REGION Network 82: [P4] Movimento BTRK da P3 Entry == a ==> P3 Exit == a ==> P3 to P4
   RUNG wire#powerrail
      Contact( #CIn.P3.Fermi.Rest )
      Contact( #Sts.P3.Fermi.Sens_Out )
      "BTrk_Presence"(Item := "BTrk".A0301."B"["BTRK_A0301_Pos3_Entry"])
      "BTrk_Absence"(Item := "BTrk".A0301."B"["BTRK_A0301_Pos3_Exit"])
      Move(in := "BTrk".A0301."B"["BTRK_A0301_Pos3_Entry"], out1 => "BTrk".A0301."B"["BTRK_A0301_Pos3_Exit"])
      "BTrk_Presence"(Item := "BTrk".A0301."B"["BTRK_A0301_Pos3_Exit"])
      Move(in := "BTrk".Empty, out1 => "BTrk".A0301."B"["BTRK_A0301_Pos3_Entry"])
   END_RUNG
   RUNG wire#powerrail
      Contact( "Sys".ByPass )
      Contact( #CIn.P3.Fermi.Rest )
      I_Contact( #Sts.P3.Fermi.Sens_Ing )
      I_Contact( #Sts.P3.Fermi.Sens_Out )
      "BTrk_Presence"(Item := "BTrk".A0301."B"["BTRK_A0301_Pos3_Entry"])
      "BTrk_Absence"(Item := "BTrk".A0301."B"["BTRK_A0301_Pos3_to_Pos4"])
      "BTrk_Absence"(Item := "BTrk".A0301."B"["BTRK_A0301_Pos4_Entry"])
      Move(in := "BTrk".A0301."B"["BTRK_A0301_Pos3_Entry"], out1 => "BTrk".A0301."B"["BTRK_A0301_Pos3_Exit"])
      "BTrk_Presence"(Item := "BTrk".A0301."B"["BTRK_A0301_Pos3_Exit"])
      Move(in := "BTrk".Empty, out1 => "BTrk".A0301."B"["BTRK_A0301_Pos3_Entry"])
   END_RUNG
   RUNG wire#powerrail
      Contact( #CIn.P3.Fermi.Rest )
      I_Contact( #Sts.P3.Fermi.Sens_Ing )
      I_Contact( #Sts.P3.Fermi.Sens_Out )
      "BTrk_Presence"(Item := "BTrk".A0301."B"["BTRK_A0301_Pos3_Exit"])
      Move(in := "BTrk".A0301."B"["BTRK_A0301_Pos3_Exit"], out1 => "BTrk".A0301."B"["BTRK_A0301_Pos3_to_Pos4"])
      "BTrk_Presence"(Item := "BTrk".A0301."B"["BTRK_A0301_Pos3_to_Pos4"])
      Move(in := "BTrk".Empty, out1 => "BTrk".A0301."B"["BTRK_A0301_Pos3_Exit"])
   END_RUNG
   // the same network as SCL:
   "BTrk_Presence"(EN := #CIn.P3.Fermi.Rest AND #Sts.P3.Fermi.Sens_Out,
                   Item := "BTrk".A0301."B"["BTRK_A0301_Pos3_Entry"],
                   ENO => #_w1);
   "BTrk_Absence"(EN := #_w1, Item := "BTrk".A0301."B"["BTRK_A0301_Pos3_Exit"], ENO => #_w2);
   IF #_w2 THEN
       "BTrk".A0301."B"["BTRK_A0301_Pos3_Exit"] := "BTrk".A0301."B"["BTRK_A0301_Pos3_Entry"];
   END_IF;
   "BTrk_Presence"(EN := #_w2, Item := "BTrk".A0301."B"["BTRK_A0301_Pos3_Exit"], ENO => #_w3);
   IF #_w3 THEN "BTrk".A0301."B"["BTRK_A0301_Pos3_Entry"] := "BTrk".Empty; END_IF;
   "BTrk_Presence"(EN := "Sys".ByPass AND #CIn.P3.Fermi.Rest AND NOT #Sts.P3.Fermi.Sens_Ing AND NOT #Sts.P3.Fermi.Sens_Out,
                   Item := "BTrk".A0301."B"["BTRK_A0301_Pos3_Entry"],
                   ENO => #_w4);
   "BTrk_Absence"(EN := #_w4, Item := "BTrk".A0301."B"["BTRK_A0301_Pos3_to_Pos4"], ENO => #_w5);
   "BTrk_Absence"(EN := #_w5, Item := "BTrk".A0301."B"["BTRK_A0301_Pos4_Entry"], ENO => #_w6);
   IF #_w6 THEN
       "BTrk".A0301."B"["BTRK_A0301_Pos3_Exit"] := "BTrk".A0301."B"["BTRK_A0301_Pos3_Entry"];
   END_IF;
   "BTrk_Presence"(EN := #_w6, Item := "BTrk".A0301."B"["BTRK_A0301_Pos3_Exit"], ENO => #_w7);
   IF #_w7 THEN "BTrk".A0301."B"["BTRK_A0301_Pos3_Entry"] := "BTrk".Empty; END_IF;
   "BTrk_Presence"(EN := #CIn.P3.Fermi.Rest AND NOT #Sts.P3.Fermi.Sens_Ing AND NOT #Sts.P3.Fermi.Sens_Out,
                   Item := "BTrk".A0301."B"["BTRK_A0301_Pos3_Exit"],
                   ENO => #_w8);
   IF #_w8 THEN
       "BTrk".A0301."B"["BTRK_A0301_Pos3_to_Pos4"] := "BTrk".A0301."B"["BTRK_A0301_Pos3_Exit"];
   END_IF;
   "BTrk_Presence"(EN := #_w8, Item := "BTrk".A0301."B"["BTRK_A0301_Pos3_to_Pos4"], ENO => #_w9);
   IF #_w9 THEN "BTrk".A0301."B"["BTRK_A0301_Pos3_Exit"] := "BTrk".Empty; END_IF;
END_REGION

REGION Network 83: [P4] Movimento BTRK da P3 a P4 == a ==> P4 Entry
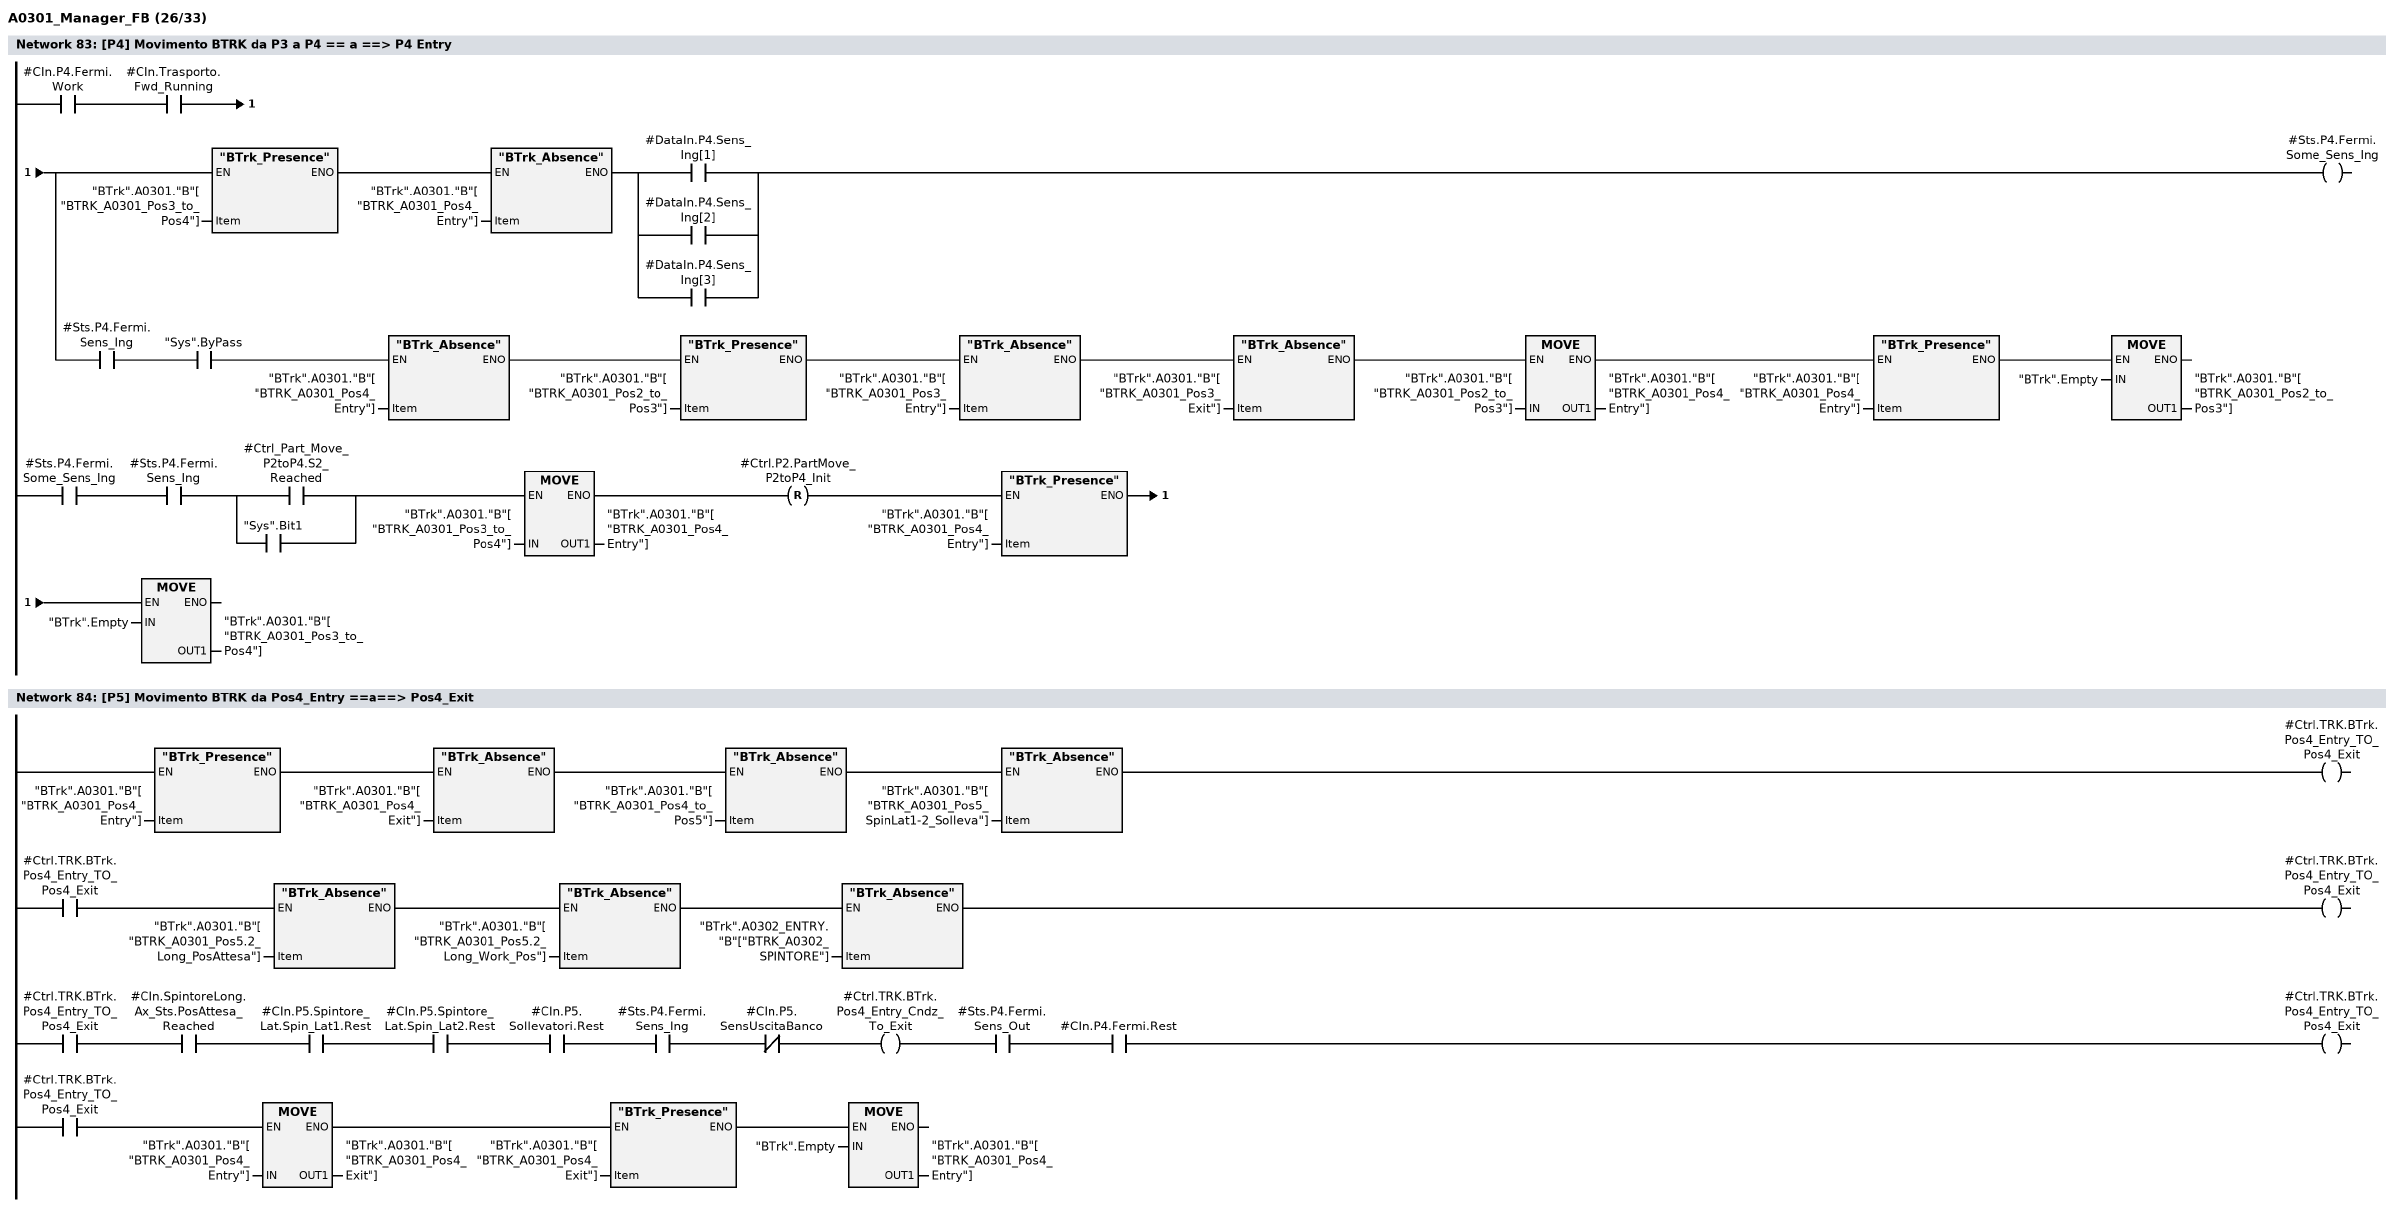
   RUNG wire#powerrail
      Contact( #CIn.P4.Fermi.Work )
      Contact( #CIn.Trasporto.Fwd_Running )
      wire#w1
      "BTrk_Presence"(Item := "BTrk".A0301."B"["BTRK_A0301_Pos3_to_Pos4"])
      "BTrk_Absence"(Item := "BTrk".A0301."B"["BTRK_A0301_Pos4_Entry"])
      wire#w2
      Contact( #DataIn.P4.Sens_Ing[1] )
      wire#w3
      Coil( #Sts.P4.Fermi.Some_Sens_Ing )
   END_RUNG
   RUNG wire#w2
      Contact( #DataIn.P4.Sens_Ing[2] )
   END_RUNG wire#w3
   RUNG wire#w2
      Contact( #DataIn.P4.Sens_Ing[3] )
   END_RUNG wire#w3
   RUNG wire#w1
      Contact( #Sts.P4.Fermi.Sens_Ing )
      Contact( "Sys".ByPass )
      "BTrk_Absence"(Item := "BTrk".A0301."B"["BTRK_A0301_Pos4_Entry"])
      "BTrk_Presence"(Item := "BTrk".A0301."B"["BTRK_A0301_Pos2_to_Pos3"])
      "BTrk_Absence"(Item := "BTrk".A0301."B"["BTRK_A0301_Pos3_Entry"])
      "BTrk_Absence"(Item := "BTrk".A0301."B"["BTRK_A0301_Pos3_Exit"])
      Move(in := "BTrk".A0301."B"["BTRK_A0301_Pos2_to_Pos3"], out1 => "BTrk".A0301."B"["BTRK_A0301_Pos4_Entry"])
      "BTrk_Presence"(Item := "BTrk".A0301."B"["BTRK_A0301_Pos4_Entry"])
      Move(in := "BTrk".Empty, out1 => "BTrk".A0301."B"["BTRK_A0301_Pos2_to_Pos3"])
   END_RUNG
   RUNG wire#powerrail
      Contact( #Sts.P4.Fermi.Some_Sens_Ing )
      Contact( #Sts.P4.Fermi.Sens_Ing )
      wire#w4
      Contact( #Ctrl_Part_Move_P2toP4.S2_Reached )
      wire#w5
      Move(in := "BTrk".A0301."B"["BTRK_A0301_Pos3_to_Pos4"], out1 => "BTrk".A0301."B"["BTRK_A0301_Pos4_Entry"])
      R_Coil( #Ctrl.P2.PartMove_P2toP4_Init )
      "BTrk_Presence"(Item := "BTrk".A0301."B"["BTRK_A0301_Pos4_Entry"])
      Move(in := "BTrk".Empty, out1 => "BTrk".A0301."B"["BTRK_A0301_Pos3_to_Pos4"])
   END_RUNG
   RUNG wire#w4
      Contact( "Sys".Bit1 )
   END_RUNG wire#w5
   // the same network as SCL:
   #_w1 := #CIn.P4.Fermi.Work AND #CIn.Trasporto.Fwd_Running;
   "BTrk_Presence"(EN := #_w1, Item := "BTrk".A0301."B"["BTRK_A0301_Pos3_to_Pos4"], ENO => #_w2);
   "BTrk_Absence"(EN := #_w2, Item := "BTrk".A0301."B"["BTRK_A0301_Pos4_Entry"], ENO => #_w3);
   #Sts.P4.Fermi.Some_Sens_Ing := #_w3 AND (#DataIn.P4.Sens_Ing[1] OR #DataIn.P4.Sens_Ing[2] OR #DataIn.P4.Sens_Ing[3]);
   "BTrk_Absence"(EN := #_w1 AND #Sts.P4.Fermi.Sens_Ing AND "Sys".ByPass,
                  Item := "BTrk".A0301."B"["BTRK_A0301_Pos4_Entry"],
                  ENO => #_w4);
   "BTrk_Presence"(EN := #_w4, Item := "BTrk".A0301."B"["BTRK_A0301_Pos2_to_Pos3"], ENO => #_w5);
   "BTrk_Absence"(EN := #_w5, Item := "BTrk".A0301."B"["BTRK_A0301_Pos3_Entry"], ENO => #_w6);
   "BTrk_Absence"(EN := #_w6, Item := "BTrk".A0301."B"["BTRK_A0301_Pos3_Exit"], ENO => #_w7);
   IF #_w7 THEN
       "BTrk".A0301."B"["BTRK_A0301_Pos4_Entry"] := "BTrk".A0301."B"["BTRK_A0301_Pos2_to_Pos3"];
   END_IF;
   "BTrk_Presence"(EN := #_w7, Item := "BTrk".A0301."B"["BTRK_A0301_Pos4_Entry"], ENO => #_w8);
   IF #_w8 THEN "BTrk".A0301."B"["BTRK_A0301_Pos2_to_Pos3"] := "BTrk".Empty; END_IF;
   IF #Sts.P4.Fermi.Some_Sens_Ing AND #Sts.P4.Fermi.Sens_Ing AND (#Ctrl_Part_Move_P2toP4.S2_Reached OR "Sys".Bit1) THEN
       "BTrk".A0301."B"["BTRK_A0301_Pos4_Entry"] := "BTrk".A0301."B"["BTRK_A0301_Pos3_to_Pos4"];
       #Ctrl.P2.PartMove_P2toP4_Init := FALSE;
   END_IF;
   "BTrk_Presence"(EN := #Sts.P4.Fermi.Some_Sens_Ing AND #Sts.P4.Fermi.Sens_Ing AND (#Ctrl_Part_Move_P2toP4.S2_Reached OR "Sys".Bit1),
                   Item := "BTrk".A0301."B"["BTRK_A0301_Pos4_Entry"],
                   ENO => #_w9);
   IF #_w9 THEN "BTrk".A0301."B"["BTRK_A0301_Pos3_to_Pos4"] := "BTrk".Empty; END_IF;
END_REGION

REGION Network 84: [P5] Movimento BTRK da Pos4_Entry ==a==> Pos4_Exit
   RUNG wire#powerrail
      "BTrk_Presence"(Item := "BTrk".A0301."B"["BTRK_A0301_Pos4_Entry"])
      "BTrk_Absence"(Item := "BTrk".A0301."B"["BTRK_A0301_Pos4_Exit"])
      "BTrk_Absence"(Item := "BTrk".A0301."B"["BTRK_A0301_Pos4_to_Pos5"])
      "BTrk_Absence"(Item := "BTrk".A0301."B"["BTRK_A0301_Pos5_SpinLat1-2_Solleva"])
      Coil( #Ctrl.TRK.BTrk.Pos4_Entry_TO_Pos4_Exit )
   END_RUNG
   RUNG wire#powerrail
      Contact( #Ctrl.TRK.BTrk.Pos4_Entry_TO_Pos4_Exit )
      "BTrk_Absence"(Item := "BTrk".A0301."B"["BTRK_A0301_Pos5.2_Long_PosAttesa"])
      "BTrk_Absence"(Item := "BTrk".A0301."B"["BTRK_A0301_Pos5.2_Long_Work_Pos"])
      "BTrk_Absence"(Item := "BTrk".A0302_ENTRY."B"["BTRK_A0302_SPINTORE"])
      Coil( #Ctrl.TRK.BTrk.Pos4_Entry_TO_Pos4_Exit )
   END_RUNG
   RUNG wire#powerrail
      Contact( #Ctrl.TRK.BTrk.Pos4_Entry_TO_Pos4_Exit )
      Contact( #CIn.SpintoreLong.Ax_Sts.PosAttesa_Reached )
      Contact( #CIn.P5.Spintore_Lat.Spin_Lat1.Rest )
      Contact( #CIn.P5.Spintore_Lat.Spin_Lat2.Rest )
      Contact( #CIn.P5.Sollevatori.Rest )
      Contact( #Sts.P4.Fermi.Sens_Ing )
      I_Contact( #CIn.P5.SensUscitaBanco )
      Coil( #Ctrl.TRK.BTrk.Pos4_Entry_Cndz_To_Exit )
      Contact( #Sts.P4.Fermi.Sens_Out )
      Contact( #CIn.P4.Fermi.Rest )
      Coil( #Ctrl.TRK.BTrk.Pos4_Entry_TO_Pos4_Exit )
   END_RUNG
   RUNG wire#powerrail
      Contact( #Ctrl.TRK.BTrk.Pos4_Entry_TO_Pos4_Exit )
      Move(in := "BTrk".A0301."B"["BTRK_A0301_Pos4_Entry"], out1 => "BTrk".A0301."B"["BTRK_A0301_Pos4_Exit"])
      "BTrk_Presence"(Item := "BTrk".A0301."B"["BTRK_A0301_Pos4_Exit"])
      Move(in := "BTrk".Empty, out1 => "BTrk".A0301."B"["BTRK_A0301_Pos4_Entry"])
   END_RUNG
   // the same network as SCL:
   "BTrk_Presence"(Item := "BTrk".A0301."B"["BTRK_A0301_Pos4_Entry"], ENO => #_w1);
   "BTrk_Absence"(EN := #_w1, Item := "BTrk".A0301."B"["BTRK_A0301_Pos4_Exit"], ENO => #_w2);
   "BTrk_Absence"(EN := #_w2, Item := "BTrk".A0301."B"["BTRK_A0301_Pos4_to_Pos5"], ENO => #_w3);
   "BTrk_Absence"(EN := #_w3, Item := "BTrk".A0301."B"["BTRK_A0301_Pos5_SpinLat1-2_Solleva"], ENO => #_w4);
   #Ctrl.TRK.BTrk.Pos4_Entry_TO_Pos4_Exit := #_w4;
   "BTrk_Absence"(EN := #Ctrl.TRK.BTrk.Pos4_Entry_TO_Pos4_Exit,
                  Item := "BTrk".A0301."B"["BTRK_A0301_Pos5.2_Long_PosAttesa"],
                  ENO => #_w5);
   "BTrk_Absence"(EN := #_w5, Item := "BTrk".A0301."B"["BTRK_A0301_Pos5.2_Long_Work_Pos"], ENO => #_w6);
   "BTrk_Absence"(EN := #_w6, Item := "BTrk".A0302_ENTRY."B"["BTRK_A0302_SPINTORE"], ENO => #_w7);
   #Ctrl.TRK.BTrk.Pos4_Entry_TO_Pos4_Exit := #_w7;
   #Ctrl.TRK.BTrk.Pos4_Entry_Cndz_To_Exit := #Ctrl.TRK.BTrk.Pos4_Entry_TO_Pos4_Exit AND #CIn.SpintoreLong.Ax_Sts.PosAttesa_Reached AND #CIn.P5.Spintore_Lat.Spin_Lat1.Rest AND #CIn.P5.Spintore_Lat.Spin_Lat2.Rest AND #CIn.P5.Sollevatori.Rest AND #Sts.P4.Fermi.Sens_Ing AND NOT #CIn.P5.SensUscitaBanco;
   #Ctrl.TRK.BTrk.Pos4_Entry_TO_Pos4_Exit := #Ctrl.TRK.BTrk.Pos4_Entry_Cndz_To_Exit AND #Sts.P4.Fermi.Sens_Out AND #CIn.P4.Fermi.Rest;
   IF #Ctrl.TRK.BTrk.Pos4_Entry_TO_Pos4_Exit THEN
       "BTrk".A0301."B"["BTRK_A0301_Pos4_Exit"] := "BTrk".A0301."B"["BTRK_A0301_Pos4_Entry"];
   END_IF;
   "BTrk_Presence"(EN := #Ctrl.TRK.BTrk.Pos4_Entry_TO_Pos4_Exit,
                   Item := "BTrk".A0301."B"["BTRK_A0301_Pos4_Exit"],
                   ENO => #_w8);
   IF #_w8 THEN "BTrk".A0301."B"["BTRK_A0301_Pos4_Entry"] := "BTrk".Empty; END_IF;
END_REGION

REGION Network 85: [P5] Movimento BTRK da Pos.4 Exit ==a==> Pos4_to_Pos5
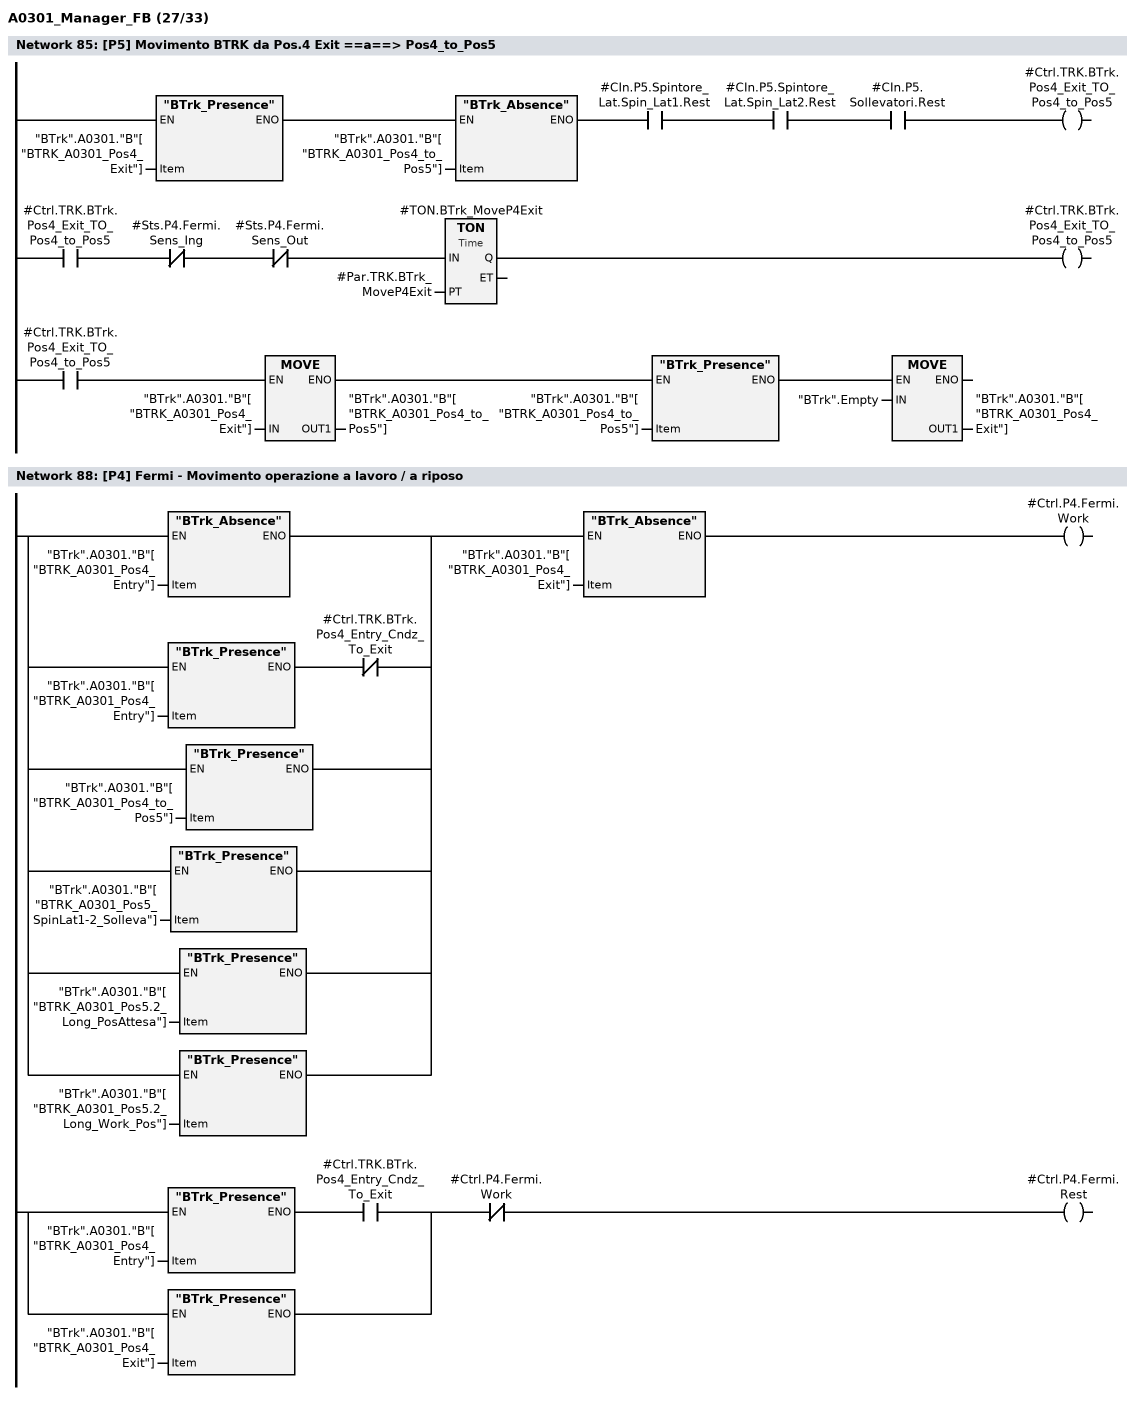
   RUNG wire#powerrail
      "BTrk_Presence"(Item := "BTrk".A0301."B"["BTRK_A0301_Pos4_Exit"])
      "BTrk_Absence"(Item := "BTrk".A0301."B"["BTRK_A0301_Pos4_to_Pos5"])
      Contact( #CIn.P5.Spintore_Lat.Spin_Lat1.Rest )
      Contact( #CIn.P5.Spintore_Lat.Spin_Lat2.Rest )
      Contact( #CIn.P5.Sollevatori.Rest )
      Coil( #Ctrl.TRK.BTrk.Pos4_Exit_TO_Pos4_to_Pos5 )
   END_RUNG
   RUNG wire#powerrail
      Contact( #Ctrl.TRK.BTrk.Pos4_Exit_TO_Pos4_to_Pos5 )
      I_Contact( #Sts.P4.Fermi.Sens_Ing )
      I_Contact( #Sts.P4.Fermi.Sens_Out )
      { S7_Templates := "time_type := Time" } #TON.BTrk_MoveP4Exit.TON(pt := #Par.TRK.BTrk_MoveP4Exit, et =>)
      Coil( #Ctrl.TRK.BTrk.Pos4_Exit_TO_Pos4_to_Pos5 )
   END_RUNG
   RUNG wire#powerrail
      Contact( #Ctrl.TRK.BTrk.Pos4_Exit_TO_Pos4_to_Pos5 )
      Move(in := "BTrk".A0301."B"["BTRK_A0301_Pos4_Exit"], out1 => "BTrk".A0301."B"["BTRK_A0301_Pos4_to_Pos5"])
      "BTrk_Presence"(Item := "BTrk".A0301."B"["BTRK_A0301_Pos4_to_Pos5"])
      Move(in := "BTrk".Empty, out1 => "BTrk".A0301."B"["BTRK_A0301_Pos4_Exit"])
   END_RUNG
   // the same network as SCL:
   "BTrk_Presence"(Item := "BTrk".A0301."B"["BTRK_A0301_Pos4_Exit"], ENO => #_w1);
   "BTrk_Absence"(EN := #_w1, Item := "BTrk".A0301."B"["BTRK_A0301_Pos4_to_Pos5"], ENO => #_w2);
   #Ctrl.TRK.BTrk.Pos4_Exit_TO_Pos4_to_Pos5 := #_w2 AND #CIn.P5.Spintore_Lat.Spin_Lat1.Rest AND #CIn.P5.Spintore_Lat.Spin_Lat2.Rest AND #CIn.P5.Sollevatori.Rest;
   #TON.BTrk_MoveP4Exit.TON(IN := #Ctrl.TRK.BTrk.Pos4_Exit_TO_Pos4_to_Pos5 AND NOT #Sts.P4.Fermi.Sens_Ing AND NOT #Sts.P4.Fermi.Sens_Out,
                           PT := #Par.TRK.BTrk_MoveP4Exit);
   #Ctrl.TRK.BTrk.Pos4_Exit_TO_Pos4_to_Pos5 := #TON.BTrk_MoveP4Exit.Q;
   IF #Ctrl.TRK.BTrk.Pos4_Exit_TO_Pos4_to_Pos5 THEN
       "BTrk".A0301."B"["BTRK_A0301_Pos4_to_Pos5"] := "BTrk".A0301."B"["BTRK_A0301_Pos4_Exit"];
   END_IF;
   "BTrk_Presence"(EN := #Ctrl.TRK.BTrk.Pos4_Exit_TO_Pos4_to_Pos5,
                   Item := "BTrk".A0301."B"["BTRK_A0301_Pos4_to_Pos5"],
                   ENO => #_w3);
   IF #_w3 THEN "BTrk".A0301."B"["BTRK_A0301_Pos4_Exit"] := "BTrk".Empty; END_IF;
END_REGION

REGION Network 87: [P4] <<< GESTIONE MOVIMENTO FERMI >>
END_REGION

REGION Network 88: [P4] Fermi - Movimento operazione a lavoro / a riposo
   RUNG wire#powerrail
      "BTrk_Absence"(Item := "BTrk".A0301."B"["BTRK_A0301_Pos4_Entry"])
      wire#w1
      "BTrk_Absence"(Item := "BTrk".A0301."B"["BTRK_A0301_Pos4_Exit"])
      Coil( #Ctrl.P4.Fermi.Work )
   END_RUNG
   RUNG wire#powerrail
      "BTrk_Presence"(Item := "BTrk".A0301."B"["BTRK_A0301_Pos4_Entry"])
      I_Contact( #Ctrl.TRK.BTrk.Pos4_Entry_Cndz_To_Exit )
   END_RUNG wire#w1
   RUNG wire#powerrail
      "BTrk_Presence"(Item := "BTrk".A0301."B"["BTRK_A0301_Pos4_to_Pos5"])
   END_RUNG wire#w1
   RUNG wire#powerrail
      "BTrk_Presence"(Item := "BTrk".A0301."B"["BTRK_A0301_Pos5_SpinLat1-2_Solleva"])
   END_RUNG wire#w1
   RUNG wire#powerrail
      "BTrk_Presence"(Item := "BTrk".A0301."B"["BTRK_A0301_Pos5.2_Long_PosAttesa"])
   END_RUNG wire#w1
   RUNG wire#powerrail
      "BTrk_Presence"(Item := "BTrk".A0301."B"["BTRK_A0301_Pos5.2_Long_Work_Pos"])
   END_RUNG wire#w1
   RUNG wire#powerrail
      "BTrk_Presence"(Item := "BTrk".A0301."B"["BTRK_A0301_Pos4_Entry"])
      Contact( #Ctrl.TRK.BTrk.Pos4_Entry_Cndz_To_Exit )
      wire#w2
      I_Contact( #Ctrl.P4.Fermi.Work )
      Coil( #Ctrl.P4.Fermi.Rest )
   END_RUNG
   RUNG wire#powerrail
      "BTrk_Presence"(Item := "BTrk".A0301."B"["BTRK_A0301_Pos4_Exit"])
   END_RUNG wire#w2
   // the same network as SCL:
   "BTrk_Absence"(Item := "BTrk".A0301."B"["BTRK_A0301_Pos4_Entry"], ENO => #_w1);
   "BTrk_Presence"(Item := "BTrk".A0301."B"["BTRK_A0301_Pos4_Entry"], ENO => #_w2);
   "BTrk_Presence"(Item := "BTrk".A0301."B"["BTRK_A0301_Pos4_to_Pos5"], ENO => #_w3);
   "BTrk_Presence"(Item := "BTrk".A0301."B"["BTRK_A0301_Pos5_SpinLat1-2_Solleva"], ENO => #_w4);
   "BTrk_Presence"(Item := "BTrk".A0301."B"["BTRK_A0301_Pos5.2_Long_PosAttesa"], ENO => #_w5);
   "BTrk_Presence"(Item := "BTrk".A0301."B"["BTRK_A0301_Pos5.2_Long_Work_Pos"], ENO => #_w6);
   "BTrk_Absence"(EN := #_w1 OR (#_w2 AND NOT #Ctrl.TRK.BTrk.Pos4_Entry_Cndz_To_Exit) OR #_w3 OR #_w4 OR #_w5 OR #_w6,
                  Item := "BTrk".A0301."B"["BTRK_A0301_Pos4_Exit"],
                  ENO => #_w7);
   #Ctrl.P4.Fermi.Work := #_w7;
   "BTrk_Presence"(Item := "BTrk".A0301."B"["BTRK_A0301_Pos4_Entry"], ENO => #_w8);
   "BTrk_Presence"(Item := "BTrk".A0301."B"["BTRK_A0301_Pos4_Exit"], ENO => #_w9);
   #Ctrl.P4.Fermi.Rest := ((#_w8 AND #Ctrl.TRK.BTrk.Pos4_Entry_Cndz_To_Exit) OR #_w9) AND NOT #Ctrl.P4.Fermi.Work;
END_REGION

REGION Network 89: [P4] Fermi - COut Manager
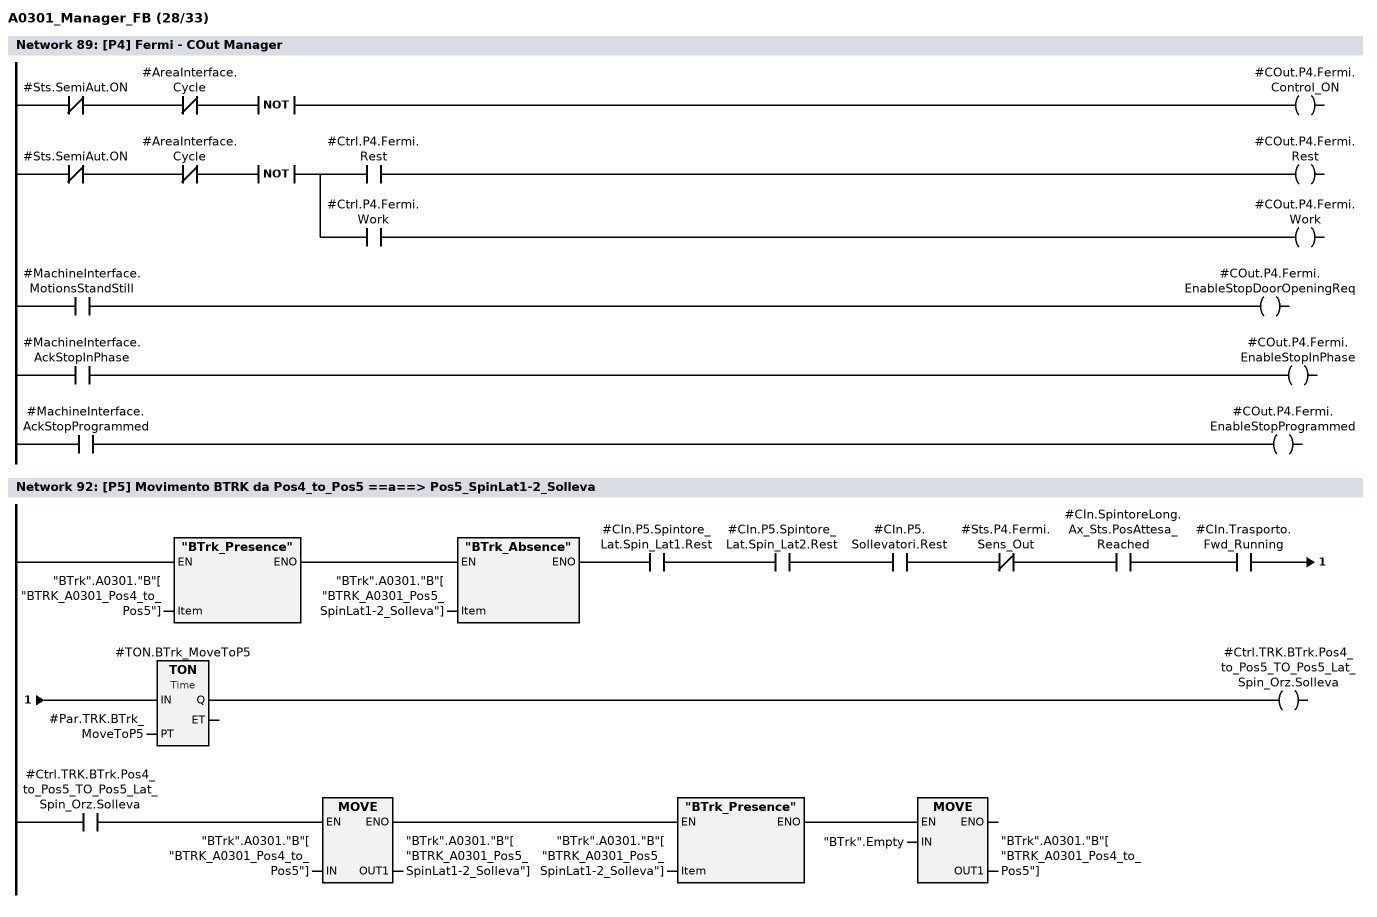
   RUNG wire#powerrail
      I_Contact( #Sts.SemiAut.ON )
      I_Contact( #AreaInterface.Cycle )
      Not()
      Coil( #COut.P4.Fermi.Control_ON )
   END_RUNG
   RUNG wire#powerrail
      I_Contact( #Sts.SemiAut.ON )
      I_Contact( #AreaInterface.Cycle )
      Not()
      wire#w1
      Contact( #Ctrl.P4.Fermi.Rest )
      Coil( #COut.P4.Fermi.Rest )
   END_RUNG
   RUNG wire#w1
      Contact( #Ctrl.P4.Fermi.Work )
      Coil( #COut.P4.Fermi.Work )
   END_RUNG
   RUNG wire#powerrail
      Contact( #MachineInterface.MotionsStandStill )
      Coil( #COut.P4.Fermi.EnableStopDoorOpeningReq )
   END_RUNG
   RUNG wire#powerrail
      Contact( #MachineInterface.AckStopInPhase )
      Coil( #COut.P4.Fermi.EnableStopInPhase )
   END_RUNG
   RUNG wire#powerrail
      Contact( #MachineInterface.AckStopProgrammed )
      Coil( #COut.P4.Fermi.EnableStopProgrammed )
   END_RUNG
   // the same network as SCL:
   #COut.P4.Fermi.Control_ON := NOT (NOT #Sts.SemiAut.ON AND NOT #AreaInterface.Cycle);
   #_w1 := NOT (NOT #Sts.SemiAut.ON AND NOT #AreaInterface.Cycle);
   #COut.P4.Fermi.Rest := #_w1 AND #Ctrl.P4.Fermi.Rest;
   #COut.P4.Fermi.Work := #_w1 AND #Ctrl.P4.Fermi.Work;
   #COut.P4.Fermi.EnableStopDoorOpeningReq := #MachineInterface.MotionsStandStill;
   #COut.P4.Fermi.EnableStopInPhase := #MachineInterface.AckStopInPhase;
   #COut.P4.Fermi.EnableStopProgrammed := #MachineInterface.AckStopProgrammed;
END_REGION

REGION Network 91: <<<<<<<<<<< POSIZIONE 5 >>>>>>>>>>>
END_REGION

REGION Network 92: [P5] Movimento BTRK da Pos4_to_Pos5 ==a==> Pos5_SpinLat1-2_Solleva
   RUNG wire#powerrail
      "BTrk_Presence"(Item := "BTrk".A0301."B"["BTRK_A0301_Pos4_to_Pos5"])
      "BTrk_Absence"(Item := "BTrk".A0301."B"["BTRK_A0301_Pos5_SpinLat1-2_Solleva"])
      Contact( #CIn.P5.Spintore_Lat.Spin_Lat1.Rest )
      Contact( #CIn.P5.Spintore_Lat.Spin_Lat2.Rest )
      Contact( #CIn.P5.Sollevatori.Rest )
      I_Contact( #Sts.P4.Fermi.Sens_Out )
      Contact( #CIn.SpintoreLong.Ax_Sts.PosAttesa_Reached )
      Contact( #CIn.Trasporto.Fwd_Running )
      { S7_Templates := "time_type := Time" } #TON.BTrk_MoveToP5.TON(pt := #Par.TRK.BTrk_MoveToP5, et =>)
      Coil( #Ctrl.TRK.BTrk.Pos4_to_Pos5_TO_Pos5_Lat_Spin_Orz.Solleva )
   END_RUNG
   RUNG wire#powerrail
      Contact( #Ctrl.TRK.BTrk.Pos4_to_Pos5_TO_Pos5_Lat_Spin_Orz.Solleva )
      Move(in := "BTrk".A0301."B"["BTRK_A0301_Pos4_to_Pos5"], out1 => "BTrk".A0301."B"["BTRK_A0301_Pos5_SpinLat1-2_Solleva"])
      "BTrk_Presence"(Item := "BTrk".A0301."B"["BTRK_A0301_Pos5_SpinLat1-2_Solleva"])
      Move(in := "BTrk".Empty, out1 => "BTrk".A0301."B"["BTRK_A0301_Pos4_to_Pos5"])
   END_RUNG
   // the same network as SCL:
   "BTrk_Presence"(Item := "BTrk".A0301."B"["BTRK_A0301_Pos4_to_Pos5"], ENO => #_w1);
   "BTrk_Absence"(EN := #_w1, Item := "BTrk".A0301."B"["BTRK_A0301_Pos5_SpinLat1-2_Solleva"], ENO => #_w2);
   #TON.BTrk_MoveToP5.TON(IN := #_w2 AND #CIn.P5.Spintore_Lat.Spin_Lat1.Rest AND #CIn.P5.Spintore_Lat.Spin_Lat2.Rest AND #CIn.P5.Sollevatori.Rest AND NOT #Sts.P4.Fermi.Sens_Out AND #CIn.SpintoreLong.Ax_Sts.PosAttesa_Reached AND #CIn.Trasporto.Fwd_Running,
                          PT := #Par.TRK.BTrk_MoveToP5);
   #Ctrl.TRK.BTrk.Pos4_to_Pos5_TO_Pos5_Lat_Spin_Orz.Solleva := #TON.BTrk_MoveToP5.Q;
   IF #Ctrl.TRK.BTrk.Pos4_to_Pos5_TO_Pos5_Lat_Spin_Orz.Solleva THEN
       "BTrk".A0301."B"["BTRK_A0301_Pos5_SpinLat1-2_Solleva"] := "BTrk".A0301."B"["BTRK_A0301_Pos4_to_Pos5"];
   END_IF;
   "BTrk_Presence"(EN := #Ctrl.TRK.BTrk.Pos4_to_Pos5_TO_Pos5_Lat_Spin_Orz.Solleva,
                   Item := "BTrk".A0301."B"["BTRK_A0301_Pos5_SpinLat1-2_Solleva"],
                   ENO => #_w3);
   IF #_w3 THEN "BTrk".A0301."B"["BTRK_A0301_Pos4_to_Pos5"] := "BTrk".Empty; END_IF;
END_REGION

REGION Network 94: [P5] <<< GESTIONE MOVIMENTO SPINTORI LATERALI - SOLLEVATORI >>>
END_REGION

REGION Network 95: [P5] Spintore Laterale - Movimento operazione a lavoro / a riposo
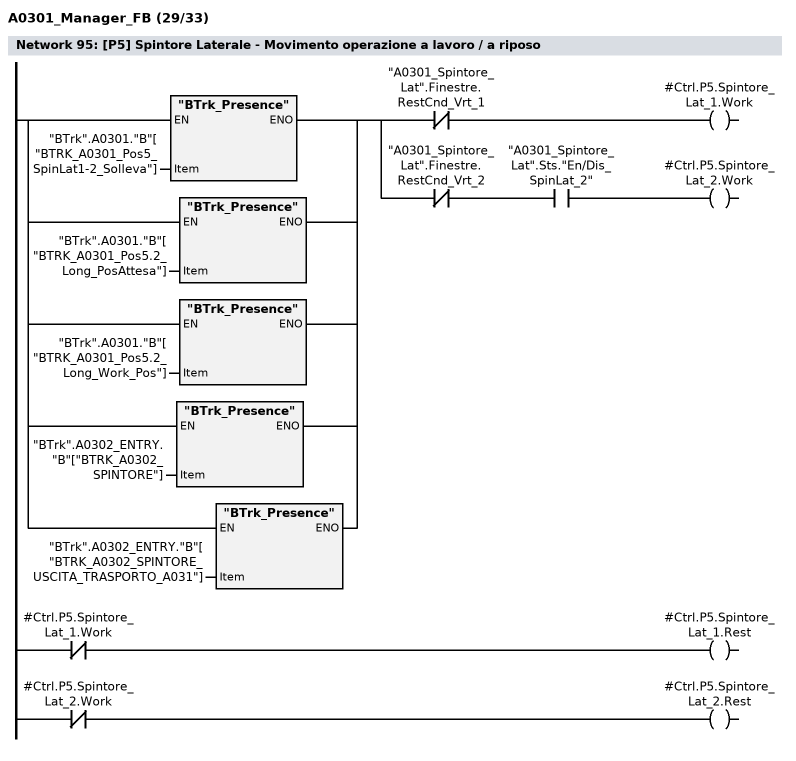
   RUNG wire#powerrail
      "BTrk_Presence"(Item := "BTrk".A0301."B"["BTRK_A0301_Pos5_SpinLat1-2_Solleva"])
      wire#w1
      I_Contact( "A0301_Spintore_Lat".Finestre.RestCnd_Vrt_1 )
      Coil( #Ctrl.P5.Spintore_Lat_1.Work )
   END_RUNG
   RUNG wire#powerrail
      "BTrk_Presence"(Item := "BTrk".A0301."B"["BTRK_A0301_Pos5.2_Long_PosAttesa"])
   END_RUNG wire#w1
   RUNG wire#powerrail
      "BTrk_Presence"(Item := "BTrk".A0301."B"["BTRK_A0301_Pos5.2_Long_Work_Pos"])
   END_RUNG wire#w1
   RUNG wire#powerrail
      "BTrk_Presence"(Item := "BTrk".A0302_ENTRY."B"["BTRK_A0302_SPINTORE"])
   END_RUNG wire#w1
   RUNG wire#powerrail
      "BTrk_Presence"(Item := "BTrk".A0302_ENTRY."B"["BTRK_A0302_SPINTORE_USCITA_TRASPORTO_A031"])
   END_RUNG wire#w1
   RUNG wire#w1
      I_Contact( "A0301_Spintore_Lat".Finestre.RestCnd_Vrt_2 )
      Contact( "A0301_Spintore_Lat".Sts."En/Dis_SpinLat_2" )
      Coil( #Ctrl.P5.Spintore_Lat_2.Work )
   END_RUNG
   RUNG wire#powerrail
      I_Contact( #Ctrl.P5.Spintore_Lat_1.Work )
      Coil( #Ctrl.P5.Spintore_Lat_1.Rest )
   END_RUNG
   RUNG wire#powerrail
      I_Contact( #Ctrl.P5.Spintore_Lat_2.Work )
      Coil( #Ctrl.P5.Spintore_Lat_2.Rest )
   END_RUNG
   // the same network as SCL:
   "BTrk_Presence"(Item := "BTrk".A0301."B"["BTRK_A0301_Pos5_SpinLat1-2_Solleva"], ENO => #_w1);
   "BTrk_Presence"(Item := "BTrk".A0301."B"["BTRK_A0301_Pos5.2_Long_PosAttesa"], ENO => #_w2);
   "BTrk_Presence"(Item := "BTrk".A0301."B"["BTRK_A0301_Pos5.2_Long_Work_Pos"], ENO => #_w3);
   "BTrk_Presence"(Item := "BTrk".A0302_ENTRY."B"["BTRK_A0302_SPINTORE"], ENO => #_w4);
   "BTrk_Presence"(Item := "BTrk".A0302_ENTRY."B"["BTRK_A0302_SPINTORE_USCITA_TRASPORTO_A031"], ENO => #_w5);
   #_w6 := #_w1 OR #_w2 OR #_w3 OR #_w4 OR #_w5;
   #Ctrl.P5.Spintore_Lat_1.Work := #_w6 AND NOT "A0301_Spintore_Lat".Finestre.RestCnd_Vrt_1;
   #Ctrl.P5.Spintore_Lat_2.Work := #_w6 AND NOT "A0301_Spintore_Lat".Finestre.RestCnd_Vrt_2 AND "A0301_Spintore_Lat".Sts."En/Dis_SpinLat_2";
   #Ctrl.P5.Spintore_Lat_1.Rest := NOT #Ctrl.P5.Spintore_Lat_1.Work;
   #Ctrl.P5.Spintore_Lat_2.Rest := NOT #Ctrl.P5.Spintore_Lat_2.Work;
END_REGION

REGION Network 96: [P5] Spintore Laterale - COut Manager
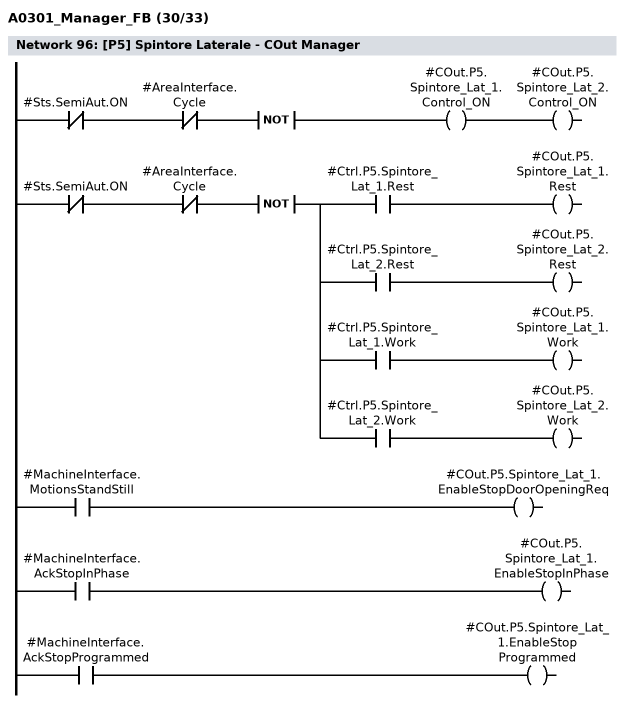
   RUNG wire#powerrail
      I_Contact( #Sts.SemiAut.ON )
      I_Contact( #AreaInterface.Cycle )
      Not()
      Coil( #COut.P5.Spintore_Lat_1.Control_ON )
      Coil( #COut.P5.Spintore_Lat_2.Control_ON )
   END_RUNG
   RUNG wire#powerrail
      I_Contact( #Sts.SemiAut.ON )
      I_Contact( #AreaInterface.Cycle )
      Not()
      wire#w1
      Contact( #Ctrl.P5.Spintore_Lat_1.Rest )
      Coil( #COut.P5.Spintore_Lat_1.Rest )
   END_RUNG
   RUNG wire#w1
      Contact( #Ctrl.P5.Spintore_Lat_2.Rest )
      Coil( #COut.P5.Spintore_Lat_2.Rest )
   END_RUNG
   RUNG wire#w1
      Contact( #Ctrl.P5.Spintore_Lat_1.Work )
      Coil( #COut.P5.Spintore_Lat_1.Work )
   END_RUNG
   RUNG wire#w1
      Contact( #Ctrl.P5.Spintore_Lat_2.Work )
      Coil( #COut.P5.Spintore_Lat_2.Work )
   END_RUNG
   RUNG wire#powerrail
      Contact( #MachineInterface.MotionsStandStill )
      Coil( #COut.P5.Spintore_Lat_1.EnableStopDoorOpeningReq )
   END_RUNG
   RUNG wire#powerrail
      Contact( #MachineInterface.AckStopInPhase )
      Coil( #COut.P5.Spintore_Lat_1.EnableStopInPhase )
   END_RUNG
   RUNG wire#powerrail
      Contact( #MachineInterface.AckStopProgrammed )
      Coil( #COut.P5.Spintore_Lat_1.EnableStopProgrammed )
   END_RUNG
   // the same network as SCL:
   #COut.P5.Spintore_Lat_1.Control_ON := NOT (NOT #Sts.SemiAut.ON AND NOT #AreaInterface.Cycle);
   #COut.P5.Spintore_Lat_2.Control_ON := #COut.P5.Spintore_Lat_1.Control_ON;
   #_w1 := NOT (NOT #Sts.SemiAut.ON AND NOT #AreaInterface.Cycle);
   #COut.P5.Spintore_Lat_1.Rest := #_w1 AND #Ctrl.P5.Spintore_Lat_1.Rest;
   #COut.P5.Spintore_Lat_2.Rest := #_w1 AND #Ctrl.P5.Spintore_Lat_2.Rest;
   #COut.P5.Spintore_Lat_1.Work := #_w1 AND #Ctrl.P5.Spintore_Lat_1.Work;
   #COut.P5.Spintore_Lat_2.Work := #_w1 AND #Ctrl.P5.Spintore_Lat_2.Work;
   #COut.P5.Spintore_Lat_1.EnableStopDoorOpeningReq := #MachineInterface.MotionsStandStill;
   #COut.P5.Spintore_Lat_1.EnableStopInPhase := #MachineInterface.AckStopInPhase;
   #COut.P5.Spintore_Lat_1.EnableStopProgrammed := #MachineInterface.AckStopProgrammed;
END_REGION

REGION Network 97: [P5] Sollevatori - Movimento operazione a lavoro / a riposo
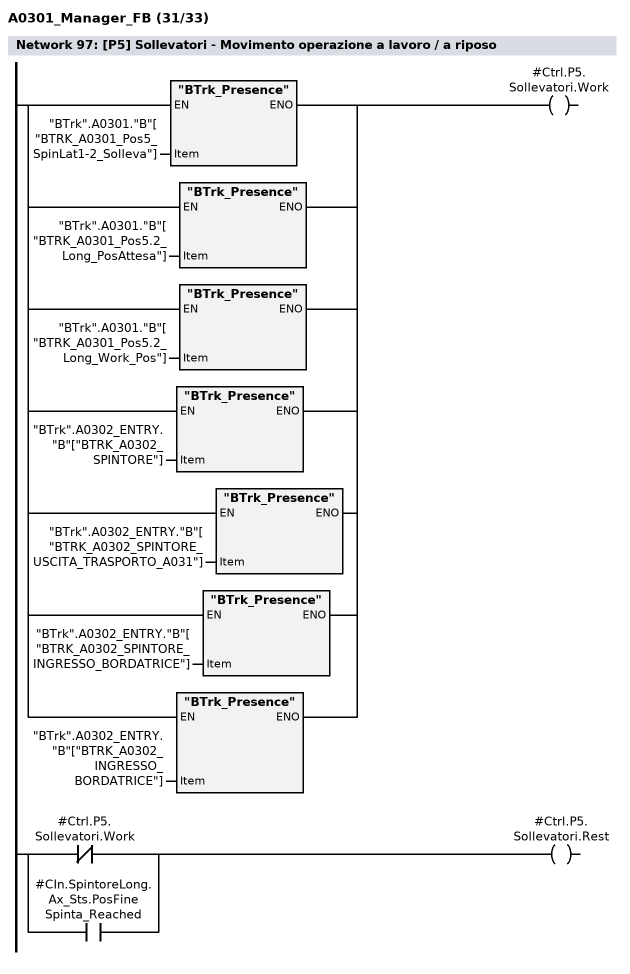
   RUNG wire#powerrail
      "BTrk_Presence"(Item := "BTrk".A0301."B"["BTRK_A0301_Pos5_SpinLat1-2_Solleva"])
      wire#w1
      Coil( #Ctrl.P5.Sollevatori.Work )
   END_RUNG
   RUNG wire#powerrail
      "BTrk_Presence"(Item := "BTrk".A0301."B"["BTRK_A0301_Pos5.2_Long_PosAttesa"])
   END_RUNG wire#w1
   RUNG wire#powerrail
      "BTrk_Presence"(Item := "BTrk".A0301."B"["BTRK_A0301_Pos5.2_Long_Work_Pos"])
   END_RUNG wire#w1
   RUNG wire#powerrail
      "BTrk_Presence"(Item := "BTrk".A0302_ENTRY."B"["BTRK_A0302_SPINTORE"])
   END_RUNG wire#w1
   RUNG wire#powerrail
      "BTrk_Presence"(Item := "BTrk".A0302_ENTRY."B"["BTRK_A0302_SPINTORE_USCITA_TRASPORTO_A031"])
   END_RUNG wire#w1
   RUNG wire#powerrail
      "BTrk_Presence"(Item := "BTrk".A0302_ENTRY."B"["BTRK_A0302_SPINTORE_INGRESSO_BORDATRICE"])
   END_RUNG wire#w1
   RUNG wire#powerrail
      "BTrk_Presence"(Item := "BTrk".A0302_ENTRY."B"["BTRK_A0302_INGRESSO_BORDATRICE"])
   END_RUNG wire#w1
   RUNG wire#powerrail
      I_Contact( #Ctrl.P5.Sollevatori.Work )
      wire#w2
      Coil( #Ctrl.P5.Sollevatori.Rest )
   END_RUNG
   RUNG wire#powerrail
      Contact( #CIn.SpintoreLong.Ax_Sts.PosFineSpinta_Reached )
   END_RUNG wire#w2
   // the same network as SCL:
   "BTrk_Presence"(Item := "BTrk".A0301."B"["BTRK_A0301_Pos5_SpinLat1-2_Solleva"], ENO => #_w1);
   "BTrk_Presence"(Item := "BTrk".A0301."B"["BTRK_A0301_Pos5.2_Long_PosAttesa"], ENO => #_w2);
   "BTrk_Presence"(Item := "BTrk".A0301."B"["BTRK_A0301_Pos5.2_Long_Work_Pos"], ENO => #_w3);
   "BTrk_Presence"(Item := "BTrk".A0302_ENTRY."B"["BTRK_A0302_SPINTORE"], ENO => #_w4);
   "BTrk_Presence"(Item := "BTrk".A0302_ENTRY."B"["BTRK_A0302_SPINTORE_USCITA_TRASPORTO_A031"], ENO => #_w5);
   "BTrk_Presence"(Item := "BTrk".A0302_ENTRY."B"["BTRK_A0302_SPINTORE_INGRESSO_BORDATRICE"], ENO => #_w6);
   "BTrk_Presence"(Item := "BTrk".A0302_ENTRY."B"["BTRK_A0302_INGRESSO_BORDATRICE"], ENO => #_w7);
   #Ctrl.P5.Sollevatori.Work := #_w1 OR #_w2 OR #_w3 OR #_w4 OR #_w5 OR #_w6 OR #_w7;
   #Ctrl.P5.Sollevatori.Rest := NOT #Ctrl.P5.Sollevatori.Work OR #CIn.SpintoreLong.Ax_Sts.PosFineSpinta_Reached;
END_REGION

REGION Network 98: [P5] Sollevatori - COut Manager
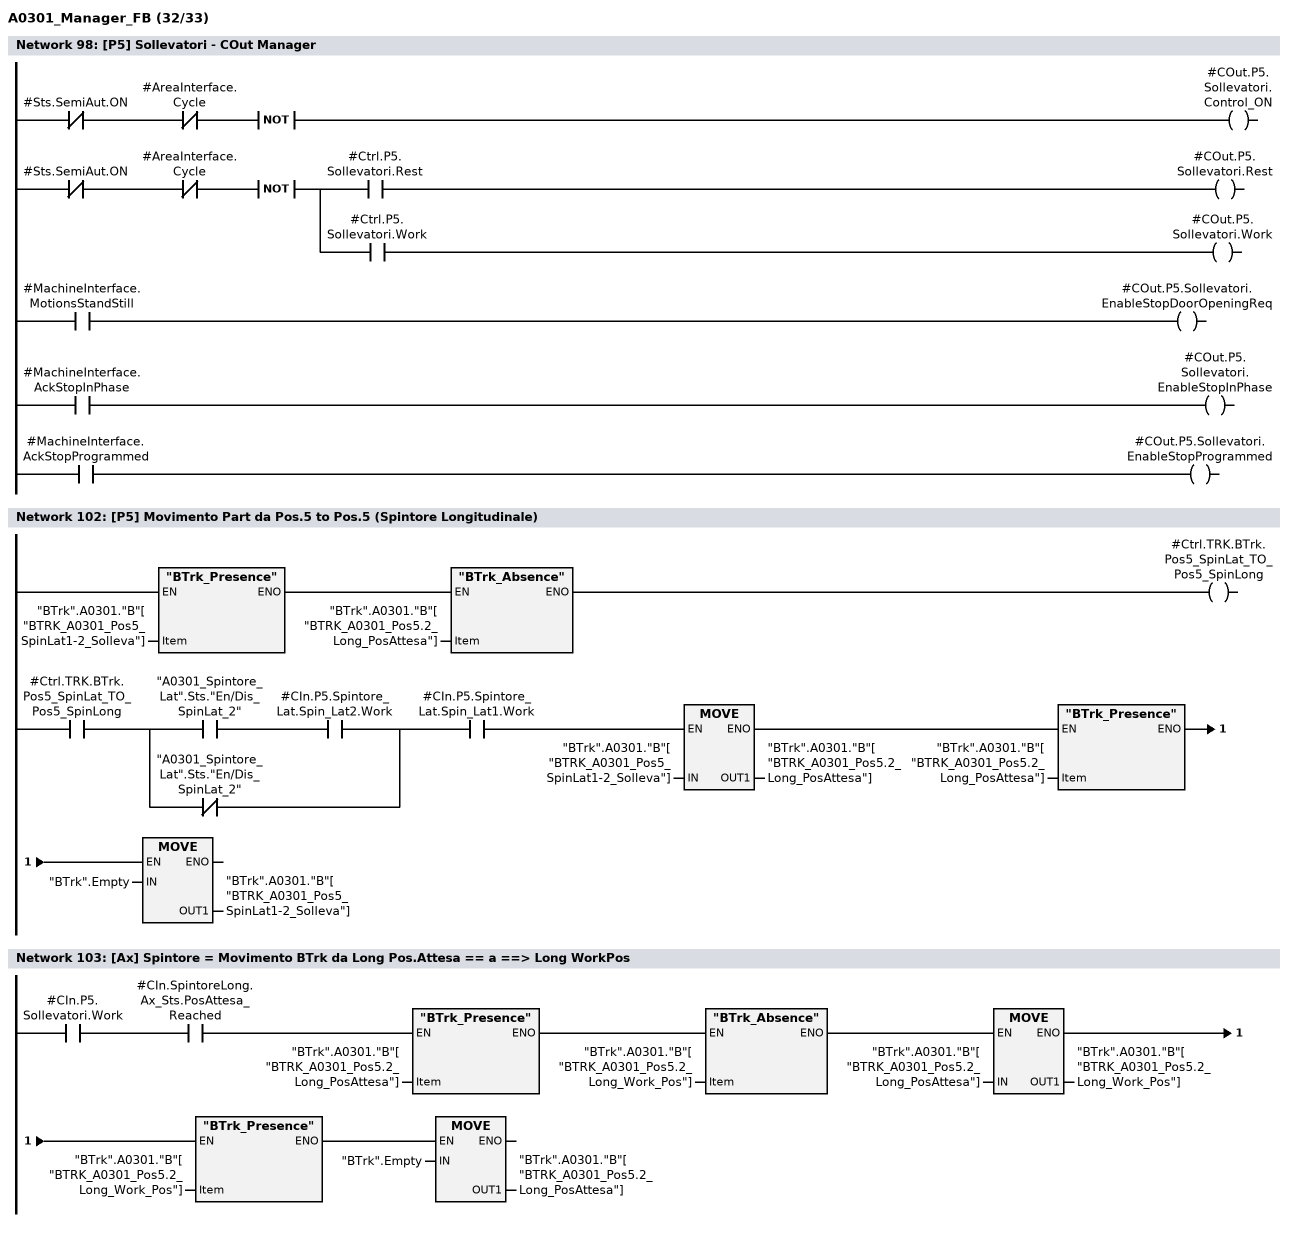
   RUNG wire#powerrail
      I_Contact( #Sts.SemiAut.ON )
      I_Contact( #AreaInterface.Cycle )
      Not()
      Coil( #COut.P5.Sollevatori.Control_ON )
   END_RUNG
   RUNG wire#powerrail
      I_Contact( #Sts.SemiAut.ON )
      I_Contact( #AreaInterface.Cycle )
      Not()
      wire#w1
      Contact( #Ctrl.P5.Sollevatori.Rest )
      Coil( #COut.P5.Sollevatori.Rest )
   END_RUNG
   RUNG wire#w1
      Contact( #Ctrl.P5.Sollevatori.Work )
      Coil( #COut.P5.Sollevatori.Work )
   END_RUNG
   RUNG wire#powerrail
      Contact( #MachineInterface.MotionsStandStill )
      Coil( #COut.P5.Sollevatori.EnableStopDoorOpeningReq )
   END_RUNG
   RUNG wire#powerrail
      Contact( #MachineInterface.AckStopInPhase )
      Coil( #COut.P5.Sollevatori.EnableStopInPhase )
   END_RUNG
   RUNG wire#powerrail
      Contact( #MachineInterface.AckStopProgrammed )
      Coil( #COut.P5.Sollevatori.EnableStopProgrammed )
   END_RUNG
   // the same network as SCL:
   #COut.P5.Sollevatori.Control_ON := NOT (NOT #Sts.SemiAut.ON AND NOT #AreaInterface.Cycle);
   #_w1 := NOT (NOT #Sts.SemiAut.ON AND NOT #AreaInterface.Cycle);
   #COut.P5.Sollevatori.Rest := #_w1 AND #Ctrl.P5.Sollevatori.Rest;
   #COut.P5.Sollevatori.Work := #_w1 AND #Ctrl.P5.Sollevatori.Work;
   #COut.P5.Sollevatori.EnableStopDoorOpeningReq := #MachineInterface.MotionsStandStill;
   #COut.P5.Sollevatori.EnableStopInPhase := #MachineInterface.AckStopInPhase;
   #COut.P5.Sollevatori.EnableStopProgrammed := #MachineInterface.AckStopProgrammed;
END_REGION

REGION Network 100: [P5] <<< GESTIONE MOVIMENTO SPINTORE LONGITUDINALE >>
END_REGION

REGION Network 102: [P5] Movimento Part da Pos.5 to Pos.5 (Spintore Longitudinale)
   RUNG wire#powerrail
      "BTrk_Presence"(Item := "BTrk".A0301."B"["BTRK_A0301_Pos5_SpinLat1-2_Solleva"])
      "BTrk_Absence"(Item := "BTrk".A0301."B"["BTRK_A0301_Pos5.2_Long_PosAttesa"])
      Coil( #Ctrl.TRK.BTrk.Pos5_SpinLat_TO_Pos5_SpinLong )
   END_RUNG
   RUNG wire#powerrail
      Contact( #Ctrl.TRK.BTrk.Pos5_SpinLat_TO_Pos5_SpinLong )
      wire#w1
      Contact( "A0301_Spintore_Lat".Sts."En/Dis_SpinLat_2" )
      Contact( #CIn.P5.Spintore_Lat.Spin_Lat2.Work )
      wire#w2
      Contact( #CIn.P5.Spintore_Lat.Spin_Lat1.Work )
      Move(in := "BTrk".A0301."B"["BTRK_A0301_Pos5_SpinLat1-2_Solleva"], out1 => "BTrk".A0301."B"["BTRK_A0301_Pos5.2_Long_PosAttesa"])
      "BTrk_Presence"(Item := "BTrk".A0301."B"["BTRK_A0301_Pos5.2_Long_PosAttesa"])
      Move(in := "BTrk".Empty, out1 => "BTrk".A0301."B"["BTRK_A0301_Pos5_SpinLat1-2_Solleva"])
   END_RUNG
   RUNG wire#w1
      I_Contact( "A0301_Spintore_Lat".Sts."En/Dis_SpinLat_2" )
   END_RUNG wire#w2
   // the same network as SCL:
   "BTrk_Presence"(Item := "BTrk".A0301."B"["BTRK_A0301_Pos5_SpinLat1-2_Solleva"], ENO => #_w1);
   "BTrk_Absence"(EN := #_w1, Item := "BTrk".A0301."B"["BTRK_A0301_Pos5.2_Long_PosAttesa"], ENO => #_w2);
   #Ctrl.TRK.BTrk.Pos5_SpinLat_TO_Pos5_SpinLong := #_w2;
   IF #Ctrl.TRK.BTrk.Pos5_SpinLat_TO_Pos5_SpinLong AND (("A0301_Spintore_Lat".Sts."En/Dis_SpinLat_2" AND #CIn.P5.Spintore_Lat.Spin_Lat2.Work) OR NOT "A0301_Spintore_Lat".Sts."En/Dis_SpinLat_2") AND #CIn.P5.Spintore_Lat.Spin_Lat1.Work THEN
       "BTrk".A0301."B"["BTRK_A0301_Pos5.2_Long_PosAttesa"] := "BTrk".A0301."B"["BTRK_A0301_Pos5_SpinLat1-2_Solleva"];
   END_IF;
   "BTrk_Presence"(EN := #Ctrl.TRK.BTrk.Pos5_SpinLat_TO_Pos5_SpinLong AND (("A0301_Spintore_Lat".Sts."En/Dis_SpinLat_2" AND #CIn.P5.Spintore_Lat.Spin_Lat2.Work) OR NOT "A0301_Spintore_Lat".Sts."En/Dis_SpinLat_2") AND #CIn.P5.Spintore_Lat.Spin_Lat1.Work,
                   Item := "BTrk".A0301."B"["BTRK_A0301_Pos5.2_Long_PosAttesa"],
                   ENO => #_w3);
   IF #_w3 THEN "BTrk".A0301."B"["BTRK_A0301_Pos5_SpinLat1-2_Solleva"] := "BTrk".Empty; END_IF;
END_REGION

REGION Network 103: [Ax] Spintore = Movimento BTrk da Long Pos.Attesa == a ==> Long WorkPos
   RUNG wire#powerrail
      Contact( #CIn.P5.Sollevatori.Work )
      Contact( #CIn.SpintoreLong.Ax_Sts.PosAttesa_Reached )
      "BTrk_Presence"(Item := "BTrk".A0301."B"["BTRK_A0301_Pos5.2_Long_PosAttesa"])
      "BTrk_Absence"(Item := "BTrk".A0301."B"["BTRK_A0301_Pos5.2_Long_Work_Pos"])
      Move(in := "BTrk".A0301."B"["BTRK_A0301_Pos5.2_Long_PosAttesa"], out1 => "BTrk".A0301."B"["BTRK_A0301_Pos5.2_Long_Work_Pos"])
      "BTrk_Presence"(Item := "BTrk".A0301."B"["BTRK_A0301_Pos5.2_Long_Work_Pos"])
      Move(in := "BTrk".Empty, out1 => "BTrk".A0301."B"["BTRK_A0301_Pos5.2_Long_PosAttesa"])
   END_RUNG
   // the same network as SCL:
   "BTrk_Presence"(EN := #CIn.P5.Sollevatori.Work AND #CIn.SpintoreLong.Ax_Sts.PosAttesa_Reached,
                   Item := "BTrk".A0301."B"["BTRK_A0301_Pos5.2_Long_PosAttesa"],
                   ENO => #_w1);
   "BTrk_Absence"(EN := #_w1, Item := "BTrk".A0301."B"["BTRK_A0301_Pos5.2_Long_Work_Pos"], ENO => #_w2);
   IF #_w2 THEN
       "BTrk".A0301."B"["BTRK_A0301_Pos5.2_Long_Work_Pos"] := "BTrk".A0301."B"["BTRK_A0301_Pos5.2_Long_PosAttesa"];
   END_IF;
   "BTrk_Presence"(EN := #_w2, Item := "BTrk".A0301."B"["BTRK_A0301_Pos5.2_Long_Work_Pos"], ENO => #_w3);
   IF #_w3 THEN "BTrk".A0301."B"["BTRK_A0301_Pos5.2_Long_PosAttesa"] := "BTrk".Empty; END_IF;
END_REGION

REGION Network 104: [P5] <<< GESTIONE MOVIMENTO SPINTORE LONGITUDINALE >>
END_REGION

REGION Network 105: <+>
END_REGION

REGION Network 106: Stop Cycle
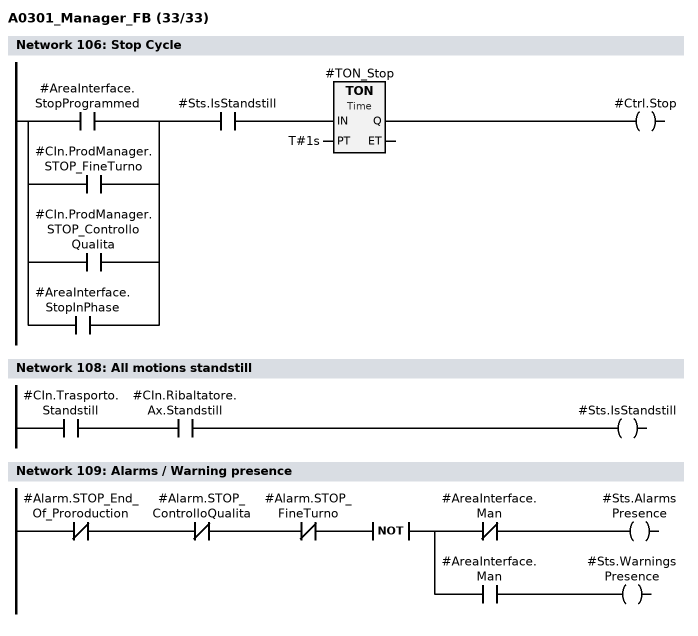
   RUNG wire#powerrail
      Contact( #AreaInterface.StopProgrammed )
      wire#w1
      Contact( #Sts.IsStandstill )
      { S7_Templates := "time_type := Time" } #TON_Stop.TON(pt := T#1s, et =>)
      Coil( #Ctrl.Stop )
   END_RUNG
   RUNG wire#powerrail
      Contact( #CIn.ProdManager.STOP_FineTurno )
   END_RUNG wire#w1
   RUNG wire#powerrail
      Contact( #CIn.ProdManager.STOP_ControlloQualita )
   END_RUNG wire#w1
   RUNG wire#powerrail
      Contact( #AreaInterface.StopInPhase )
   END_RUNG wire#w1
   // the same network as SCL:
   #TON_Stop.TON(IN := (#AreaInterface.StopProgrammed OR #CIn.ProdManager.STOP_FineTurno OR #CIn.ProdManager.STOP_ControlloQualita OR #AreaInterface.StopInPhase) AND #Sts.IsStandstill,
                 PT := T#1s);
   #Ctrl.Stop := #TON_Stop.Q;
END_REGION

REGION Network 107: << FINAL OPERATIONS >>
   // +
   // +
   // +
   // +
   // +
   // +
   // +
   // +
   // +
   // +
   // +
   // +
   // +
END_REGION

REGION Network 108: All motions standstill
   RUNG wire#powerrail
      Contact( #CIn.Trasporto.Standstill )
      Contact( #CIn.Ribaltatore.Ax.Standstill )
      Coil( #Sts.IsStandstill )
   END_RUNG
   // the same network as SCL:
   #Sts.IsStandstill := #CIn.Trasporto.Standstill AND #CIn.Ribaltatore.Ax.Standstill;
END_REGION

REGION Network 109: Alarms / Warning presence
   RUNG wire#powerrail
      I_Contact( #Alarm.STOP_End_Of_Proroduction )
      I_Contact( #Alarm.STOP_ControlloQualita )
      I_Contact( #Alarm.STOP_FineTurno )
      Not()
      wire#w1
      I_Contact( #AreaInterface.Man )
      Coil( #Sts.AlarmsPresence )
   END_RUNG
   RUNG wire#w1
      Contact( #AreaInterface.Man )
      Coil( #Sts.WarningsPresence )
   END_RUNG
   // the same network as SCL:
   #_w1 := NOT (NOT #Alarm.STOP_End_Of_Proroduction AND NOT #Alarm.STOP_ControlloQualita AND NOT #Alarm.STOP_FineTurno);
   #Sts.AlarmsPresence := #_w1 AND NOT #AreaInterface.Man;
   #Sts.WarningsPresence := #_w1 AND #AreaInterface.Man;
END_REGION

REGION Network 110 (SCL): Collect machine to area interface
   #MachineInterface.AlarmsPresence := #Sts.AlarmsPresence;

   #MachineInterface.WarningPresence := #Sts.WarningsPresence;

   #MachineInterface.MotionsStandStill := #Sts.IsStandstill;

   #MachineInterface.AutReady := #AreaInterface.Aut AND NOT #Sts.AlarmsPresence;


   #MachineInterface.AckStopInPhase := #AreaInterface.StopInPhase AND #Ctrl.Stop;

   #MachineInterface.AckStopProgrammed := #AreaInterface.StopProgrammed AND #Ctrl.Stop;


   #MachineInterface.Aborting := #AreaInterface.Aut AND #Sts.AlarmsPresence;
END_REGION
END_FUNCTION_BLOCK

FUNCTION "A0301_StopperSelSensorON" : Void
{ S7_Optimized_Access := 'TRUE' ; Published := 'FALSE' }
VERSION : 0.1
   VAR_INPUT 
      PLen : Real;
   END_VAR

   VAR_OUTPUT 
      SensorsToUse : Array[1..3] of Bool;
   END_VAR


BEGIN
	#SensorsToUse[1] := TRUE;
	#SensorsToUse[2] := TRUE;
	#SensorsToUse[3] := TRUE;
	
	IF #PLen <= "A0301_PERS".Par.CaseD_PLen_Lim AND  #PLen > "A0301_PERS".Par.CaseC_PLen_Lim THEN
	    #SensorsToUse[1] := "A0301_PERS".Par.CaseD_StopperSensor.%X0 := TRUE;
	    #SensorsToUse[2] := "A0301_PERS".Par.CaseD_StopperSensor.%X1 := TRUE;
	    #SensorsToUse[3] := "A0301_PERS".Par.CaseD_StopperSensor.%X2 := TRUE;
	    RETURN;
	END_IF;
	
	IF #PLen <= "A0301_PERS".Par.CaseC_PLen_Lim AND #PLen > "A0301_PERS".Par.CaseB_PLen_Lim THEN
	    #SensorsToUse[1] := "A0301_PERS".Par.CaseC_StopperSensor.%X0 := TRUE;
	    #SensorsToUse[2] := "A0301_PERS".Par.CaseC_StopperSensor.%X1 := TRUE;
	    #SensorsToUse[3] := "A0301_PERS".Par.CaseC_StopperSensor.%X2 := FALSE;
	    RETURN;
	END_IF;
	
	
	IF #PLen <= "A0301_PERS".Par.CaseB_PLen_Lim AND #PLen > "A0301_PERS".Par.CaseA_PLen_Lim THEN
	    #SensorsToUse[1] := "A0301_PERS".Par.CaseB_StopperSensor.%X0 := TRUE;
	    #SensorsToUse[2] := "A0301_PERS".Par.CaseB_StopperSensor.%X1 := TRUE;
	    #SensorsToUse[3] := "A0301_PERS".Par.CaseB_StopperSensor.%X2 := FALSE;
	    RETURN;
	END_IF;
	
	IF #PLen <= "A0301_PERS".Par.CaseA_PLen_Lim THEN
	    
	    #SensorsToUse[1] := "A0301_PERS".Par.CaseA_StopperSensor.%X0 := TRUE;
	    #SensorsToUse[2] := "A0301_PERS".Par.CaseA_StopperSensor.%X1 := FALSE;
	    #SensorsToUse[3] := "A0301_PERS".Par.CaseA_StopperSensor.%X2 := FALSE;
	ELSIF #PLen < "A0301_PERS".Par.CaseA_PLen_Lim THEN
	    #SensorsToUse[1] := "A0301_PERS".Par.CaseA_StopperSensor.%X0 := TRUE;
	    #SensorsToUse[2] := "A0301_PERS".Par.CaseA_StopperSensor.%X1 := FALSE;
	    #SensorsToUse[3] := "A0301_PERS".Par.CaseA_StopperSensor.%X2 := FALSE;
	    RETURN;
	END_IF;
	
	
	
	
	
END_FUNCTION

FUNCTION "A0301_Trasporto_CALL" : Void   // FC111, LAD
// stored: SetENOAutomatically false
   VAR CONSTANT
      MISSING : Int;
   END_VAR
BEGIN

REGION Network 1 (SCL): << TRASFERIMENTO stati CIn del blocco >>
   // TRASFERIMENTO #CIn MANAGER
   "A0301_Trasporto".CIn.OP_SemiAut_PB := "A0301_Manager".DataIn.SemiAut_Pb;

   // TRASFERIMENTO #CIn DRIVE
   "A0301_Trasporto".CIn.Drive.Manager := "A0301_Manager".COut.Trasporto;
END_REGION

REGION Network 2 (SCL): << TRASFERIMENTO stati DataIn >>
   // "Sys".ByPass ===> SOSTITUIRE CON INGRESSI
   // TRASFERIMENTO #DataIn STATI BUTTON TRASPORTO
   // PB TRASPORTO
   "A0301_Trasporto".DataIn.PB.Bwd_Minus := "A03_HMI".MB3.Button.A0301.Trasporto.Bwd_Minus;
   "A0301_Trasporto".DataIn.PB.Fwd_Plus := "A03_HMI".MB3.Button.A0301.Trasporto.Fwd_Plus;
END_REGION

REGION Network 3 (SCL): DSI
   //
   "A0301_Trasporto".DSI := "F_DB".DSI_Trasporto;
END_REGION

REGION Network 4 (SCL): HW
   //
   "A0301_Trasporto".HWID_Ax_TEL1 := "HW_Const_Values".CU5_PN_1480A1_1_Standard_telegram_1;
END_REGION

REGION Network 5 (SCL): Drive
   // 
   "A0301_Trasporto".Drive.Infeed_ON := "Areas_ITF".AG.Infeed_Running;;
   "A0301_Trasporto".Drive.AccessPoint := "HW_Const_Values".CU5_PN_600A1_ModuleAccessPoint;
   "A0301_Trasporto".Drive.AxisID := "CU5_ID_3_1480A1_1_1480M1";
   "A0301_Trasporto".Drive.TokenChain := "TOKENCHAIN_CU5";
END_REGION

REGION Network 6: << RICHIAMO - TRASPORTO >>
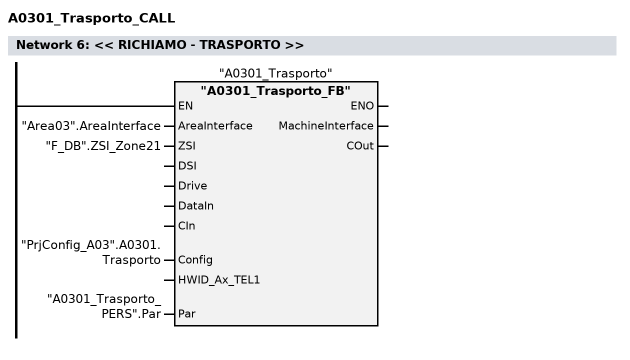
   RUNG wire#powerrail
      "A0301_Trasporto"(AreaInterface := "Area03".AreaInterface, ZSI := "F_DB".ZSI_Zone21, DSI :=, Drive :=, DataIn :=, CIn :=, Config := "PrjConfig_A03".A0301.Trasporto, HWID_Ax_TEL1 :=, Par := "A0301_Trasporto_PERS".Par, MachineInterface =>, COut =>)
   END_RUNG
   // the same network as SCL:
   "A0301_Trasporto"(AreaInterface := "Area03".AreaInterface,   // "A0301_Trasporto_FB"
                     ZSI := "F_DB".ZSI_Zone21,
                     Config := "PrjConfig_A03".A0301.Trasporto,
                     Par := "A0301_Trasporto_PERS".Par);
END_REGION
END_FUNCTION

FUNCTION_BLOCK "A0301_Trasporto_FB"   // FB61, LAD
TITLE = == GESTIONE NASTRI TRASPORTO ==
// stored: MemoryReserve 100, SetENOAutomatically false
   VAR_INPUT
      AreaInterface : "AreaInterface";
      ZSI : "udt_ZoneSafetyInterface";
      DSI : "udt_DeviceSafetyInterface";
      Drive : "TAx_DriveInterface";
      DataIn : "SpeedMachine_DataIn";
      CIn : Struct
         Drive : "SpeedMachine_CIn";
         OP_SemiAut_PB : Bool;
      END_STRUCT;
      Config : "SpeedMachine_Config";
      HWID_Ax_TEL1 : HW_SUBMODULE;
   END_VAR
   VAR_OUTPUT
      MachineInterface { ExternalAccessible := 'False'; ExternalVisible := 'False'; ExternalWritable := 'False'} : "MachineInterface";
      COut : Struct
         Ax : "SpeedMachine_COut";
         Ax_VelOveride : Struct
            Enable : Bool;
            Value : Real;
         END_STRUCT;
      END_STRUCT;
   END_VAR
   VAR_IN_OUT
      Par : Struct
         Ax : "SpeedMachine_Par";
         Ax_Aut : "A0301_Mach_Speed_Par";
      END_STRUCT;
   END_VAR
   VAR
      Alarm : Struct
         Ax { ExternalVisible := 'False'} : "SpeedMachine_Alr";
      END_STRUCT;
      Warning : Struct
         Ax { S7_SetPoint := 'True'} : "SpeedMachine_Wng";
         OP_REST_MissingCnd : Bool;   // Mancanza comando arresto
         OP_WORK_MissingCnd : Bool;   // Mancanza consenso lavoro
      END_STRUCT;
      Ax : "SpeedMachine_FB";
      ValueVelOvr { ExternalAccessible := 'False'; ExternalVisible := 'False'; ExternalWritable := 'False'} : Array[1..10] of Real;
      Sts : Struct
         OP_CanMoveFreely : Bool;
         OP_Bwd_Cnd : Bool;
         OP_Fwd_Cnd : Bool;
      END_STRUCT;
      Ctrl : Struct
         OP_Bwd_Man : Bool;
         OP_Fwd_Man : Bool;
         OP_Bwd_Aut : Bool;
         OP_Fwd_Aut : Bool;
         OP_Bwd_Run : Bool;
         OP_Fwd_Run : Bool;
      END_STRUCT;
      AUX : Struct
         OP_Bwd_PB : Bool;
         OP_Fwd_PB : Bool;
      END_STRUCT;
      TON_OP_REST_MissingCnd { S7_SetPoint := 'True'} : TON_TIME;
      TON_OP_WORK_MissingCnd { S7_SetPoint := 'True'} : TON_TIME;
   END_VAR
   VAR_TEMP
      PE : Struct
         OP_Bwd_PB : Bool;
         OP_Fwd_PB : Bool;
      END_STRUCT;
      VelOvr_Max : Real;   // Velocità max trovata
      i : Int;
      Check : Struct
         Cndz1_StartFwd : Bool;   // Check conditions to P4
         Cndz2_StartFwd : Bool;   // Check conditions to Allineatore laterale
      END_STRUCT;
   END_VAR
   VAR_TEMP   // added for the SCL form of the ladder/FBD networks
      _w1 : Bool;
      _w2 : Bool;
      _w3 : Bool;
   END_VAR
BEGIN

REGION Network 1 (SCL): == Riferimenti [Ax] - Speed Machine ==
   // ******************************************************************************************
   REGION // TRASFERIMENTO DELLE RAMPE

       // Rampe in Manuale
       IF #AreaInterface.Man AND NOT #CIn.OP_SemiAut_PB THEN
           #Ax.CIn.Manager.Vel := #Par.Ax.Man.VelFwdHigh;
           #Ax.CIn.Manager.Acc := #Par.Ax.Man.Acc;
           #Ax.CIn.Manager.Dec := #Par.Ax.Man.Dec;
       END_IF;
   END_REGION


   // ******************************************************************************************
   REGION // CALCOLO DELLA VELOCITA' TRASFERITA DALL'IMPIANTO IN BASE ALLA LUNGHEZZA DEL PEZZO 

       // Inizializzo variabile di appoggio controllo overide massimo a un valore basso rispetto setpoint
       IF "Sys".AuxFirstPLCCycle THEN
           #VelOvr_Max := 100.0;
       END_IF;

       // Trasferisco le varibili su un array
       #ValueVelOvr[1] := "PPrf_MAIN".ON_WORK.A0301_A0302.Trasporto.VelOvr_PLen_UpTo_1000;
       #ValueVelOvr[2] := "PPrf_MAIN".ON_WORK.A0301_A0302.Trasporto.VelOvr_PLen_UpTo_1500;
       #ValueVelOvr[3] := "PPrf_MAIN".ON_WORK.A0301_A0302.Trasporto.VelOvr_PLen_UpTo_2000;
       #ValueVelOvr[4] := "PPrf_MAIN".ON_WORK.A0301_A0302.Trasporto.VelOvr_PLen_UpTo_2500;
       #ValueVelOvr[5] := "PPrf_MAIN".ON_WORK.A0301_A0302.Trasporto.VelOvr_PLen_UpTo_3000;
       #ValueVelOvr[6] := "PPrf_MAIN".ON_WORK.A0301_A0302.Trasporto.VelOvr_PLen_UpTo_3500;
       #ValueVelOvr[7] := "PPrf_MAIN".ON_WORK.A0301_A0302.Trasporto.VelOvr_PLen_UpTo_4000;
       #ValueVelOvr[8] := "PPrf_MAIN".ON_WORK.A0301_A0302.Trasporto.VelOvr_PLen_UpTo_4500;
       #ValueVelOvr[9] := "PPrf_MAIN".ON_WORK.A0301_A0302.Trasporto.VelOvr_PLen_UpTo_5000;
       #ValueVelOvr[10] := "PPrf_MAIN".ON_WORK.A0301_A0302.Trasporto.VelOvr_PLen_UpTo_5500;


       // Ciclo per verificare la variabile maggiore per prenderla in lavoro
       FOR #i := 1 TO 10 DO
           IF #ValueVelOvr[#i] >= #VelOvr_Max THEN
               #VelOvr_Max := #ValueVelOvr[#i];
           END_IF;
       END_FOR;
   END_REGION ;

   IF #VelOvr_Max = 0.0 THEN
       #VelOvr_Max := 100.0;
   END_IF;

   // ******************************************************************************************
   REGION // CALCOLO DELLA VELOCITA' E TRASFERIMENTO IN BASE ALLO STATO IMPIANTO
       #Ax.CIn.Manager := #CIn.Drive.Manager;

       IF #Ax.CIn.Manager.Control_ON THEN
           // CALCOLO VELOCITA' IN BASE ALL'OVERIDE
           IF #Ax.AreaInterface.Aut THEN
               #Ax.CIn.Manager.Vel := (#Par.Ax_Aut.Aut_Vel * #VelOvr_Max);
           END_IF;

           IF #CIn.OP_SemiAut_PB AND NOT #Ax.AreaInterface.Aut THEN
               #Ax.CIn.Manager.Vel := (#Par.Ax_Aut.SemiAut_Vel* #VelOvr_Max);
               #Ax.CIn.Manager.Acc := #Par.Ax_Aut.Aut_Acc;
               #Ax.CIn.Manager.Dec := #Par.Ax_Aut.Aut_Dec;
           END_IF;
       END_IF;
   END_REGION ;
   //


       #COut.Ax_VelOveride.Enable := TRUE;
       #COut.Ax_VelOveride.Value := #VelOvr_Max;
END_REGION

REGION Network 3: Operazione può muoversi liberamente perchè non sposta nessun BEAM
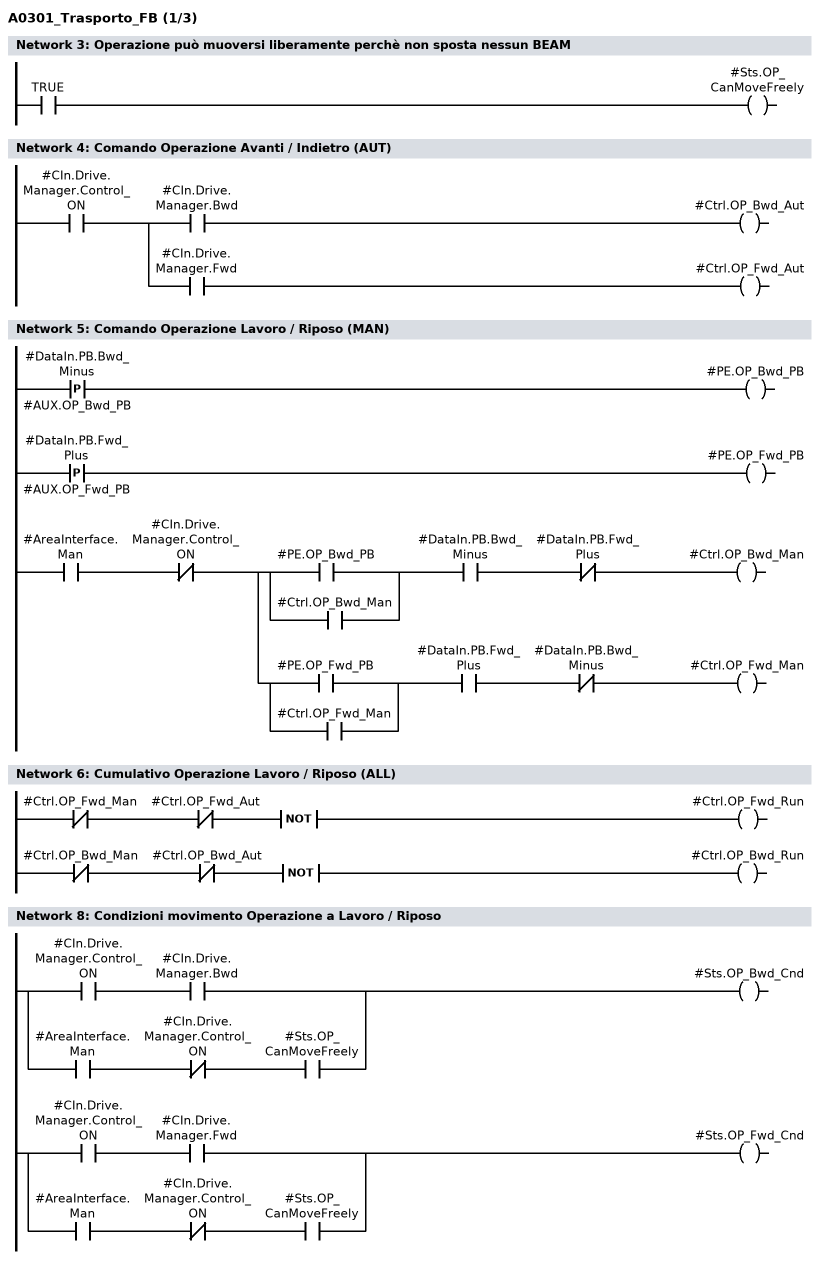
   RUNG wire#powerrail
      Contact( TRUE )
      Coil( #Sts.OP_CanMoveFreely )
   END_RUNG
   // the same network as SCL:
   #Sts.OP_CanMoveFreely := TRUE;
END_REGION

REGION Network 4: Comando Operazione Avanti / Indietro (AUT)
   RUNG wire#powerrail
      Contact( #CIn.Drive.Manager.Control_ON )
      wire#w1
      Contact( #CIn.Drive.Manager.Bwd )
      Coil( #Ctrl.OP_Bwd_Aut )
   END_RUNG
   RUNG wire#w1
      Contact( #CIn.Drive.Manager.Fwd )
      Coil( #Ctrl.OP_Fwd_Aut )
   END_RUNG
   // the same network as SCL:
   #Ctrl.OP_Bwd_Aut := #CIn.Drive.Manager.Control_ON AND #CIn.Drive.Manager.Bwd;
   #Ctrl.OP_Fwd_Aut := #CIn.Drive.Manager.Control_ON AND #CIn.Drive.Manager.Fwd;
END_REGION

REGION Network 5: Comando Operazione Lavoro / Riposo (MAN)
   RUNG wire#powerrail
      P_Contact(operand := #DataIn.PB.Bwd_Minus, bit := #AUX.OP_Bwd_PB)
      Coil( #PE.OP_Bwd_PB )
   END_RUNG
   RUNG wire#powerrail
      P_Contact(operand := #DataIn.PB.Fwd_Plus, bit := #AUX.OP_Fwd_PB)
      Coil( #PE.OP_Fwd_PB )
   END_RUNG
   RUNG wire#powerrail
      Contact( #AreaInterface.Man )
      I_Contact( #CIn.Drive.Manager.Control_ON )
      wire#w1
      Contact( #PE.OP_Bwd_PB )
      wire#w2
      Contact( #DataIn.PB.Bwd_Minus )
      I_Contact( #DataIn.PB.Fwd_Plus )
      Coil( #Ctrl.OP_Bwd_Man )
   END_RUNG
   RUNG wire#w1
      Contact( #Ctrl.OP_Bwd_Man )
   END_RUNG wire#w2
   RUNG wire#w1
      Contact( #PE.OP_Fwd_PB )
      wire#w3
      Contact( #DataIn.PB.Fwd_Plus )
      I_Contact( #DataIn.PB.Bwd_Minus )
      Coil( #Ctrl.OP_Fwd_Man )
   END_RUNG
   RUNG wire#w1
      Contact( #Ctrl.OP_Fwd_Man )
   END_RUNG wire#w3
   // the same network as SCL:
   #_w1 := #DataIn.PB.Bwd_Minus AND NOT #AUX.OP_Bwd_PB;   // rising edge of #DataIn.PB.Bwd_Minus
   #AUX.OP_Bwd_PB := #DataIn.PB.Bwd_Minus;
   #PE.OP_Bwd_PB := #_w1;
   #_w2 := #DataIn.PB.Fwd_Plus AND NOT #AUX.OP_Fwd_PB;   // rising edge of #DataIn.PB.Fwd_Plus
   #AUX.OP_Fwd_PB := #DataIn.PB.Fwd_Plus;
   #PE.OP_Fwd_PB := #_w2;
   #_w3 := #AreaInterface.Man AND NOT #CIn.Drive.Manager.Control_ON;
   #Ctrl.OP_Bwd_Man := #_w3 AND (#PE.OP_Bwd_PB OR #Ctrl.OP_Bwd_Man) AND #DataIn.PB.Bwd_Minus AND NOT #DataIn.PB.Fwd_Plus;
   #Ctrl.OP_Fwd_Man := #_w3 AND (#PE.OP_Fwd_PB OR #Ctrl.OP_Fwd_Man) AND #DataIn.PB.Fwd_Plus AND NOT #DataIn.PB.Bwd_Minus;
END_REGION

REGION Network 6: Cumulativo Operazione Lavoro / Riposo (ALL)
   RUNG wire#powerrail
      I_Contact( #Ctrl.OP_Fwd_Man )
      I_Contact( #Ctrl.OP_Fwd_Aut )
      Not()
      Coil( #Ctrl.OP_Fwd_Run )
   END_RUNG
   RUNG wire#powerrail
      I_Contact( #Ctrl.OP_Bwd_Man )
      I_Contact( #Ctrl.OP_Bwd_Aut )
      Not()
      Coil( #Ctrl.OP_Bwd_Run )
   END_RUNG
   // the same network as SCL:
   #Ctrl.OP_Fwd_Run := NOT (NOT #Ctrl.OP_Fwd_Man AND NOT #Ctrl.OP_Fwd_Aut);
   #Ctrl.OP_Bwd_Run := NOT (NOT #Ctrl.OP_Bwd_Man AND NOT #Ctrl.OP_Bwd_Aut);
END_REGION

REGION Network 7: <+>
END_REGION

REGION Network 8: Condizioni movimento Operazione a Lavoro / Riposo
   RUNG wire#powerrail
      Contact( #CIn.Drive.Manager.Control_ON )
      Contact( #CIn.Drive.Manager.Bwd )
      wire#w1
      Coil( #Sts.OP_Bwd_Cnd )
   END_RUNG
   RUNG wire#powerrail
      Contact( #AreaInterface.Man )
      I_Contact( #CIn.Drive.Manager.Control_ON )
      Contact( #Sts.OP_CanMoveFreely )
   END_RUNG wire#w1
   RUNG wire#powerrail
      Contact( #CIn.Drive.Manager.Control_ON )
      Contact( #CIn.Drive.Manager.Fwd )
      wire#w2
      Coil( #Sts.OP_Fwd_Cnd )
   END_RUNG
   RUNG wire#powerrail
      Contact( #AreaInterface.Man )
      I_Contact( #CIn.Drive.Manager.Control_ON )
      Contact( #Sts.OP_CanMoveFreely )
   END_RUNG wire#w2
   // the same network as SCL:
   #Sts.OP_Bwd_Cnd := (#CIn.Drive.Manager.Control_ON AND #CIn.Drive.Manager.Bwd) OR (#AreaInterface.Man AND NOT #CIn.Drive.Manager.Control_ON AND #Sts.OP_CanMoveFreely);
   #Sts.OP_Fwd_Cnd := (#CIn.Drive.Manager.Control_ON AND #CIn.Drive.Manager.Fwd) OR (#AreaInterface.Man AND NOT #CIn.Drive.Manager.Control_ON AND #Sts.OP_CanMoveFreely);
END_REGION

REGION Network 9 (SCL): [Ax] Cin Manager Comando arresto / lavoro
   //
   #Ax.CIn.Manager.Bwd := FALSE;
   //************************************
   #Ax.CIn.Manager.Fwd := FALSE;
   //
   // CIn Manager  Control ON se ho un richiesta di comando attiva
   #Ax.CIn.Manager.Control_ON := #Ctrl.OP_Fwd_Run OR #Ctrl.OP_Bwd_Run;

   // CIn Manager Frw se ho un richiesta di comando arresto attiva
   #Ax.CIn.Manager.Fwd := #Ctrl.OP_Fwd_Run AND #Sts.OP_Fwd_Cnd ;

   // CIn Manager Brw se ho un richiesta di comando arresto attiva
   #Ax.CIn.Manager.Bwd := #Ctrl.OP_Bwd_Run AND #Sts.OP_Bwd_Cnd;
END_REGION

REGION Network 10 (SCL): [Ax] CIn Abilitazioni Stop Manager
   // CIn Manager Stop per richiesta apertura safety
   // 
   #Ax.CIn.Manager.EnableStopDoorOpeningReq := #CIn.Drive.Manager.EnableStopDoorOpeningReq;

   // CIn Manager Stop in fase delle macchine precedenti
   // 
   #Ax.CIn.Manager.EnableStopInPhase := #CIn.Drive.Manager.EnableStopInPhase;

   // CIn Manager Stop programmato configurabile a piacere
   // 
   #Ax.CIn.Manager.EnableStopProgrammed := #CIn.Drive.Manager.EnableStopProgrammed;
END_REGION

REGION Network 11: <+>
END_REGION

REGION Network 12: Warning manacanza condizioni esecuzione Operazione RIPOSO / LAVORO
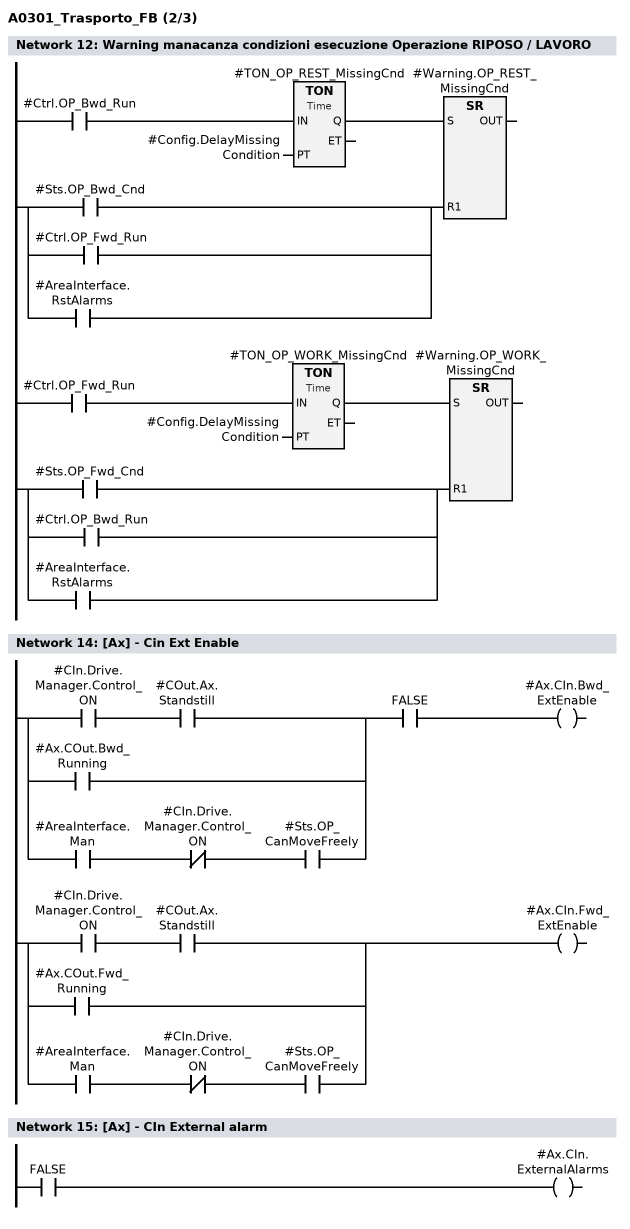
   RUNG wire#powerrail
      Contact( #Ctrl.OP_Bwd_Run )
      { S7_Templates := "time_type := Time" } #TON_OP_REST_MissingCnd.TON(pt := #Config.DelayMissingCondition, et =>)
      S_SR(operand := #Warning.OP_REST_MissingCnd, r1 := wire#w1)
   END_RUNG
   RUNG wire#powerrail
      Contact( #Sts.OP_Bwd_Cnd )
   END_RUNG wire#w1
   RUNG wire#powerrail
      Contact( #Ctrl.OP_Fwd_Run )
   END_RUNG wire#w1
   RUNG wire#powerrail
      Contact( #AreaInterface.RstAlarms )
   END_RUNG wire#w1
   RUNG wire#powerrail
      Contact( #Ctrl.OP_Fwd_Run )
      { S7_Templates := "time_type := Time" } #TON_OP_WORK_MissingCnd.TON(pt := #Config.DelayMissingCondition, et =>)
      S_SR(operand := #Warning.OP_WORK_MissingCnd, r1 := wire#w2)
   END_RUNG
   RUNG wire#powerrail
      Contact( #Sts.OP_Fwd_Cnd )
   END_RUNG wire#w2
   RUNG wire#powerrail
      Contact( #Ctrl.OP_Bwd_Run )
   END_RUNG wire#w2
   RUNG wire#powerrail
      Contact( #AreaInterface.RstAlarms )
   END_RUNG wire#w2
   // the same network as SCL:
   #TON_OP_REST_MissingCnd(IN := #Ctrl.OP_Bwd_Run, PT := #Config.DelayMissingCondition);   // TON
   IF #TON_OP_REST_MissingCnd.Q THEN
       #Warning.OP_REST_MissingCnd := TRUE;   // SR flip-flop
   END_IF;
   IF #Sts.OP_Bwd_Cnd OR #Ctrl.OP_Fwd_Run OR #AreaInterface.RstAlarms THEN
       #Warning.OP_REST_MissingCnd := FALSE;
   END_IF;
   #TON_OP_WORK_MissingCnd(IN := #Ctrl.OP_Fwd_Run, PT := #Config.DelayMissingCondition);   // TON
   IF #TON_OP_WORK_MissingCnd.Q THEN
       #Warning.OP_WORK_MissingCnd := TRUE;   // SR flip-flop
   END_IF;
   IF #Sts.OP_Fwd_Cnd OR #Ctrl.OP_Bwd_Run OR #AreaInterface.RstAlarms THEN
       #Warning.OP_WORK_MissingCnd := FALSE;
   END_IF;
END_REGION

REGION Network 13: <+>
END_REGION

REGION Network 14: [Ax] - Cin Ext Enable
   RUNG wire#powerrail
      Contact( #CIn.Drive.Manager.Control_ON )
      Contact( #COut.Ax.Standstill )
      wire#w1
      Contact( FALSE )
      Coil( #Ax.CIn.Bwd_ExtEnable )
   END_RUNG
   RUNG wire#powerrail
      Contact( #Ax.COut.Bwd_Running )
   END_RUNG wire#w1
   RUNG wire#powerrail
      Contact( #AreaInterface.Man )
      I_Contact( #CIn.Drive.Manager.Control_ON )
      Contact( #Sts.OP_CanMoveFreely )
   END_RUNG wire#w1
   RUNG wire#powerrail
      Contact( #CIn.Drive.Manager.Control_ON )
      Contact( #COut.Ax.Standstill )
      wire#w2
      Coil( #Ax.CIn.Fwd_ExtEnable )
   END_RUNG
   RUNG wire#powerrail
      Contact( #Ax.COut.Fwd_Running )
   END_RUNG wire#w2
   RUNG wire#powerrail
      Contact( #AreaInterface.Man )
      I_Contact( #CIn.Drive.Manager.Control_ON )
      Contact( #Sts.OP_CanMoveFreely )
   END_RUNG wire#w2
   // the same network as SCL:
   #Ax.CIn.Bwd_ExtEnable := ((#CIn.Drive.Manager.Control_ON AND #COut.Ax.Standstill) OR #Ax.COut.Bwd_Running OR (#AreaInterface.Man AND NOT #CIn.Drive.Manager.Control_ON AND #Sts.OP_CanMoveFreely)) AND FALSE;
   #Ax.CIn.Fwd_ExtEnable := (#CIn.Drive.Manager.Control_ON AND #COut.Ax.Standstill) OR #Ax.COut.Fwd_Running OR (#AreaInterface.Man AND NOT #CIn.Drive.Manager.Control_ON AND #Sts.OP_CanMoveFreely);
END_REGION

REGION Network 15: [Ax] - CIn External alarm
   RUNG wire#powerrail
      Contact( FALSE )
      Coil( #Ax.CIn.ExternalAlarms )
   END_RUNG
   // the same network as SCL:
   #Ax.CIn.ExternalAlarms := FALSE;
END_REGION

REGION Network 16: <+>
END_REGION

REGION Network 17: [Ax] - SpeedMachine
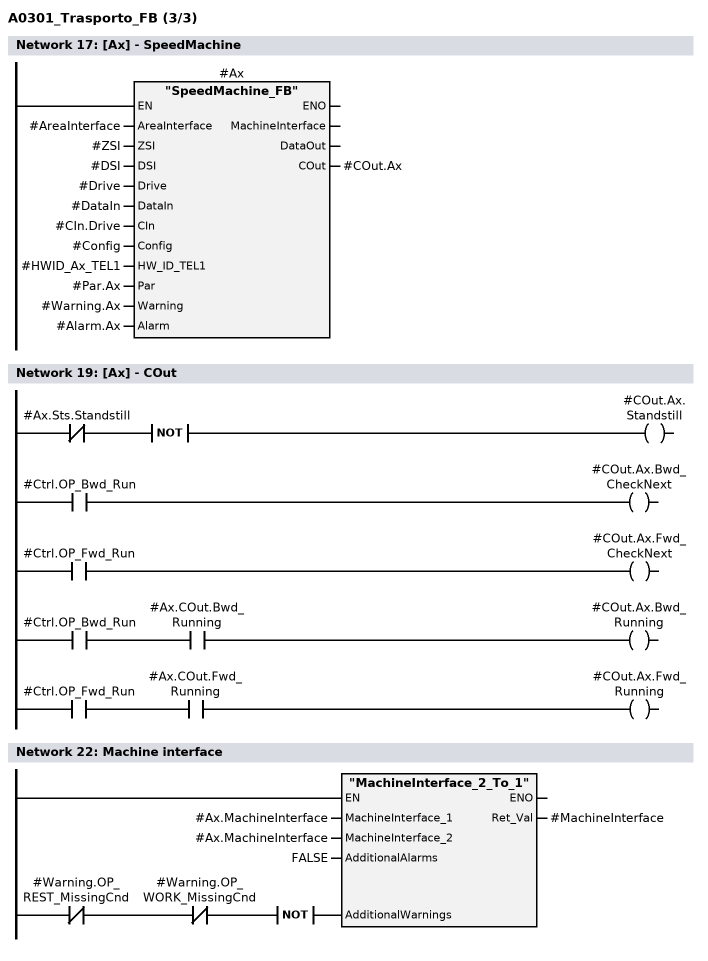
   RUNG wire#powerrail
      #Ax(AreaInterface := #AreaInterface, ZSI := #ZSI, DSI := #DSI, Drive := #Drive, DataIn := #DataIn, CIn := #CIn.Drive, Config := #Config, HW_ID_TEL1 := #HWID_Ax_TEL1, Par := #Par.Ax, Warning := #Warning.Ax, Alarm := #Alarm.Ax, MachineInterface =>, DataOut =>, COut => #COut.Ax)
   END_RUNG
   // the same network as SCL:
   #Ax(AreaInterface := #AreaInterface,   // "SpeedMachine_FB"
       ZSI := #ZSI,
       DSI := #DSI,
       Drive := #Drive,
       DataIn := #DataIn,
       CIn := #CIn.Drive,
       Config := #Config,
       HW_ID_TEL1 := #HWID_Ax_TEL1,
       Par := #Par.Ax,
       Warning := #Warning.Ax,
       Alarm := #Alarm.Ax,
       COut => #COut.Ax);
END_REGION

REGION Network 18: <+>
END_REGION

REGION Network 19: [Ax] - COut
   RUNG wire#powerrail
      I_Contact( #Ax.Sts.Standstill )
      Not()
      Coil( #COut.Ax.Standstill )
   END_RUNG
   RUNG wire#powerrail
      Contact( #Ctrl.OP_Bwd_Run )
      Coil( #COut.Ax.Bwd_CheckNext )
   END_RUNG
   RUNG wire#powerrail
      Contact( #Ctrl.OP_Fwd_Run )
      Coil( #COut.Ax.Fwd_CheckNext )
   END_RUNG
   RUNG wire#powerrail
      Contact( #Ctrl.OP_Bwd_Run )
      Contact( #Ax.COut.Bwd_Running )
      Coil( #COut.Ax.Bwd_Running )
   END_RUNG
   RUNG wire#powerrail
      Contact( #Ctrl.OP_Fwd_Run )
      Contact( #Ax.COut.Fwd_Running )
      Coil( #COut.Ax.Fwd_Running )
   END_RUNG
   // the same network as SCL:
   #COut.Ax.Standstill := NOT (NOT #Ax.Sts.Standstill);
   #COut.Ax.Bwd_CheckNext := #Ctrl.OP_Bwd_Run;
   #COut.Ax.Fwd_CheckNext := #Ctrl.OP_Fwd_Run;
   #COut.Ax.Bwd_Running := #Ctrl.OP_Bwd_Run AND #Ax.COut.Bwd_Running;
   #COut.Ax.Fwd_Running := #Ctrl.OP_Fwd_Run AND #Ax.COut.Fwd_Running;
END_REGION

REGION Network 21: << MAIN MACHINE STATUS >>
END_REGION

REGION Network 22: Machine interface
   RUNG wire#powerrail
      "MachineInterface_2_To_1"(AdditionalWarnings := wire#w1, MachineInterface_1 := #Ax.MachineInterface, MachineInterface_2 := #Ax.MachineInterface, AdditionalAlarms := FALSE, Ret_Val => #MachineInterface)
   END_RUNG
   RUNG wire#powerrail
      I_Contact( #Warning.OP_REST_MissingCnd )
      I_Contact( #Warning.OP_WORK_MissingCnd )
      Not()
   END_RUNG wire#w1
   // the same network as SCL:
   #MachineInterface := "MachineInterface_2_To_1"(MachineInterface_1 := #Ax.MachineInterface,
                           MachineInterface_2 := #Ax.MachineInterface,
                           AdditionalAlarms := FALSE,
                           AdditionalWarnings := NOT (NOT #Warning.OP_REST_MissingCnd AND NOT #Warning.OP_WORK_MissingCnd));
END_REGION
END_FUNCTION_BLOCK

FUNCTION "A0301_Fermi_P1_CALL" : Void   // FC117, LAD
// stored: SetENOAutomatically false
BEGIN

REGION Network 1 (SCL): << TRASFERIMENTO stati CIn del blocco >>
   // TRASFERIMENTO #CIn MANAGER
   "A0301_Fermi_P1".CIn.Manager_Fermi := "A0301_Manager".COut.P1.Fermi;
   "A0301_Fermi_P1".CIn.Manager_Paregg := "A0301_Manager".COut.P1.Pareggiatore;
   //
   "A0301_Fermi_P1".CIn.SemiAut := "A0301_Manager".DataIn.SemiAut_Pb;

   // Trasferimento condizione di start Sfalsatore
   // 
   "A0301_Fermi_P1".CIn.P1.Cndz_Pareggiatore := "A0301_Manager".Ctrl.P1.Pareggiatore.Work;

   // Trasferimenti status lettura posizioni Trasporto al Cin delle stazioni
   "A0301_Fermi_P1".CIn.Trasporto := "A0301_Trasporto".COut.Ax;
END_REGION

REGION Network 2 (SCL): << TRASFERIMENTO stati DataIn >>
   // SOSTITUIRE SYS.BYPASS

   REGION TRASFERIMENTO DataIn DIGITAL INPUT dei LIMIT SWITCH

       // Trasferimento ingressi digitali Limit Switch Fermi P1
       // 
       "A0301_Fermi_P1".Fermi[1].DataIn.Rest_Ls[1] := "A0301_CinghiaTrasporto_1.1_Ls_Rest_3";
       "A0301_Fermi_P1".Fermi[2].DataIn.Rest_Ls[1] := "A0301_CinghiaTrasporto_2.1_Ls_Rest_3";
       "A0301_Fermi_P1".Fermi[3].DataIn.Rest_Ls[1] := "A0301_CinghiaTrasporto_3.1_Ls_Rest_3";
       "A0301_Fermi_P1".Fermi[4].DataIn.Rest_Ls[1] := "A0301_CinghiaTrasporto_4.1_Ls_Rest_3";
       "A0301_Fermi_P1".Fermi[5].DataIn.Rest_Ls[1] := "A0301_CinghiaTrasporto_5.1_Ls_Rest_3";
       "A0301_Fermi_P1".Fermi[6].DataIn.Rest_Ls[1] := "A0301_CinghiaTrasporto_6.1_Ls_Rest_3";

       // Trasferimento ingressi digitali Limit Switch Sfalsatore P1
       "A0301_Fermi_P1".Pareggiatore.DataIn.Rest_Ls[1] := "A0301_Pareggiatore_Ls_Rest";
       "A0301_Fermi_P1".Pareggiatore.DataIn.Work_Ls[1] :=  "A0301_Pareggiatore_Ls_Work";
       //
   END_REGION ;
END_REGION

REGION Network 3: DataIn - Fermi
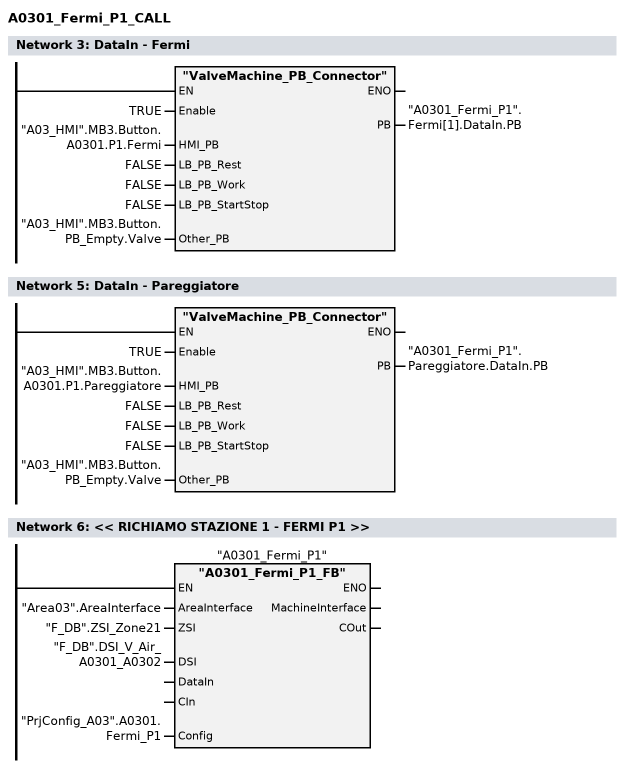
   RUNG wire#powerrail
      "ValveMachine_PB_Connector"(Enable := TRUE, HMI_PB := "A03_HMI".MB3.Button.A0301.P1.Fermi, LB_PB_Rest := FALSE, LB_PB_Work := FALSE, LB_PB_StartStop := FALSE, Other_PB := "A03_HMI".MB3.Button.PB_Empty.Valve, PB => "A0301_Fermi_P1".Fermi[1].DataIn.PB)
   END_RUNG
   // the same network as SCL:
   "ValveMachine_PB_Connector"(Enable := TRUE,
                           HMI_PB := "A03_HMI".MB3.Button.A0301.P1.Fermi,
                           LB_PB_Rest := FALSE,
                           LB_PB_Work := FALSE,
                           LB_PB_StartStop := FALSE,
                           Other_PB := "A03_HMI".MB3.Button.PB_Empty.Valve,
                           PB => "A0301_Fermi_P1".Fermi[1].DataIn.PB);
END_REGION

REGION Network 4 (SCL): DataIn - Fermi [1..6]
   // TRASFERIMENTO STATO PULSANTI - Comando manuale diretto 
   "A0301_Fermi_P1".Fermi[6].DataIn.PB.Rest := "A0301_Fermi_P1".Fermi[5].DataIn.PB.Rest := "A0301_Fermi_P1".Fermi[4].DataIn.PB.Rest :=
   "A0301_Fermi_P1".Fermi[3].DataIn.PB.Rest := "A0301_Fermi_P1".Fermi[2].DataIn.PB.Rest := "A0301_Fermi_P1".Fermi[1].DataIn.PB.Rest;

   "A0301_Fermi_P1".Fermi[6].DataIn.PB.Work := "A0301_Fermi_P1".Fermi[5].DataIn.PB.Work := "A0301_Fermi_P1".Fermi[4].DataIn.PB.Work :=
   "A0301_Fermi_P1".Fermi[3].DataIn.PB.Work := "A0301_Fermi_P1".Fermi[2].DataIn.PB.Work := "A0301_Fermi_P1".Fermi[1].DataIn.PB.Work;
END_REGION

REGION Network 5: DataIn - Pareggiatore
   RUNG wire#powerrail
      "ValveMachine_PB_Connector"(Enable := TRUE, HMI_PB := "A03_HMI".MB3.Button.A0301.P1.Pareggiatore, LB_PB_Rest := FALSE, LB_PB_Work := FALSE, LB_PB_StartStop := FALSE, Other_PB := "A03_HMI".MB3.Button.PB_Empty.Valve, PB => "A0301_Fermi_P1".Pareggiatore.DataIn.PB)
   END_RUNG
   // the same network as SCL:
   "ValveMachine_PB_Connector"(Enable := TRUE,
                           HMI_PB := "A03_HMI".MB3.Button.A0301.P1.Pareggiatore,
                           LB_PB_Rest := FALSE,
                           LB_PB_Work := FALSE,
                           LB_PB_StartStop := FALSE,
                           Other_PB := "A03_HMI".MB3.Button.PB_Empty.Valve,
                           PB => "A0301_Fermi_P1".Pareggiatore.DataIn.PB);
END_REGION

REGION Network 6: << RICHIAMO STAZIONE 1 - FERMI P1 >>
   RUNG wire#powerrail
      "A0301_Fermi_P1"(AreaInterface := "Area03".AreaInterface, ZSI := "F_DB".ZSI_Zone21, DSI := "F_DB".DSI_V_Air_A0301_A0302, DataIn :=, CIn :=, Config := "PrjConfig_A03".A0301.Fermi_P1, MachineInterface =>, COut =>)
   END_RUNG
   // the same network as SCL:
   "A0301_Fermi_P1"(AreaInterface := "Area03".AreaInterface,   // "A0301_Fermi_P1_FB"
                    ZSI := "F_DB".ZSI_Zone21,
                    DSI := "F_DB".DSI_V_Air_A0301_A0302,
                    Config := "PrjConfig_A03".A0301.Fermi_P1);
END_REGION

REGION Network 7 (SCL): << TRASFERIMENTO stati DataOut >>
   REGION COMANDO DELLE USCITE FERMI P1

       // Fermi blocco prodotto Stazione P1 - RIPOSO
       // 
       "A0301_CinghiaTrasporto_1.1_V_Rest_3":= "A0301_Fermi_P1".Fermi[1].DataOut.RestSolenoid;
       "A0301_CinghiaTrasporto_2.1_V_Rest_3" := "A0301_Fermi_P1".Fermi[2].DataOut.RestSolenoid;
       "A0301_CinghiaTrasporto_3.1_V_Rest_3" := "A0301_Fermi_P1".Fermi[3].DataOut.RestSolenoid;
       "A0301_CinghiaTrasporto_4.1_V_Rest_3" := "A0301_Fermi_P1".Fermi[4].DataOut.RestSolenoid;
       "A0301_CinghiaTrasporto_5.1_V_Rest_3" := "A0301_Fermi_P1".Fermi[5].DataOut.RestSolenoid;
       "A0301_CinghiaTrasporto_6.1_V_Rest_3" := "A0301_Fermi_P1".Fermi[6].DataOut.RestSolenoid;

       // Fermi blocco prodotto Stazione P1 - LAVORO
       // 
       "A0301_CinghiaTrasporto_1.1_V_Work_4" := "A0301_Fermi_P1".Fermi[1].DataOut.WorkSolenoid;
       "A0301_CinghiaTrasporto_2.1_V_Work_4" := "A0301_Fermi_P1".Fermi[2].DataOut.WorkSolenoid;
       "A0301_CinghiaTrasporto_3.1_V_Work_4" := "A0301_Fermi_P1".Fermi[3].DataOut.WorkSolenoid;
       "A0301_CinghiaTrasporto_4.1_V_Work_4" := "A0301_Fermi_P1".Fermi[4].DataOut.WorkSolenoid;
       "A0301_CinghiaTrasporto_5.1_V_Work_4" := "A0301_Fermi_P1".Fermi[5].DataOut.WorkSolenoid;
       "A0301_CinghiaTrasporto_6.1_V_Work_4" := "A0301_Fermi_P1".Fermi[6].DataOut.WorkSolenoid;
   END_REGION ;

   REGION COMANDO DELLE USCITE SFALSATORE P1
       // Sfasatore Semi guscio prodotto Stazione P1 - RIPOSO
       // 
       "A0301_Pareggiatore_V_Rest" := "A0301_Fermi_P1".Pareggiatore.DataOut.RestSolenoid;

       // Sfasatore Semi guscio prodotto Stazione P1 - LAVORO
       // 
       "A0301_Pareggiatore_V_Work" := "A0301_Fermi_P1".Pareggiatore.DataOut.WorkSolenoid;
   END_REGION ;
END_REGION
END_FUNCTION

FUNCTION_BLOCK "A0301_Fermi_P1_FB"   // FB89, LAD
TITLE = == GESTIONE DELLA STAZIONE P1 ==
// stored: MemoryReserve 100, SetENOAutomatically false
   VAR_INPUT
      AreaInterface : "AreaInterface";
      ZSI : "udt_ZoneSafetyInterface";
      DSI : "udt_DeviceSafetyInterface";
      DataIn : Struct
         OP_Rest_PB : Bool;
         OP_Work_PB : Bool;
      END_STRUCT;
      CIn : Struct
         Manager_Fermi : "ValveMachine_Manager";
         Manager_Paregg : "ValveMachine_Manager";
         SemiAut : Bool;
         P1 : Struct
            Cndz_Sfalsatore : Bool;
            Cndz_Pareggiatore : Bool;
         END_STRUCT;
         Trasporto : "SpeedMachine_COut";
      END_STRUCT;
      Config : Struct
         Fermi : Array[1..6] of "ValveMachine_Config";
         Pareggiatore : "ValveMachine_Config";
         DelayMissingCondition : Time := T#3s;
      END_STRUCT;
   END_VAR
   VAR_OUTPUT
      MachineInterface : "MachineInterface";
      COut : Struct
         Fermi : "ValveMachine_COut";
         Pareggiatore : "ValveMachine_COut";
      END_STRUCT;
   END_VAR
   VAR
      Alarm : Struct
         Fermi : Array[1..6] of "ValveAlr";
         Pareggiatore { S7_SetPoint := 'True'} : "ValveAlr";
      END_STRUCT;
      Warning : Struct
         OP_REST_MissingCnd : Bool;   // Mancanza comando arresto
         OP_WORK_MissingCnd : Bool;   // Mancanza consenso lavoro
         Fermi : Array[1..6] of "ValveMachine_Wng";
         Pareggiatore { S7_SetPoint := 'True'} : "ValveMachine_Wng";
      END_STRUCT;
      HMI : Struct
         Selection : Array[1..6] of Bool;   // 0=Disable / 1=Enable Pin
         FermiSts { S7_SetPoint := 'True'} : "UDT_HMI-Sts_ValvePosA0301";
         PareggiatoreSts { S7_SetPoint := 'True'} : "UDT_HMI-Sts_ValvePosA0301";
         B_ResetShiftDone : Bool;
      END_STRUCT;
      Sts : Struct
         Fermi_AlarmPresence : Bool;
         OP_CanMoveFreely : Bool;
         OP_Rest_Cnd : Bool;
         Op_Work_Cnd : Bool;
      END_STRUCT;
      Ctrl : Struct
         OP_Rest_Man : Bool;
         OP_Work_Man : Bool;
         OP_Rest_Aut : Bool;
         OP_Work_Aut : Bool;
         OP_Rest : Bool;
         OP_Work : Bool;
      END_STRUCT;
      Fermi : Array[1..6] of "ValveMachine_FB";
      Pareggiatore { S7_SetPoint := 'True'} : "ValveMachine_FB";
      AUX : Struct
         OP_Rest_PB : Bool;
         OP_Work_PB : Bool;
      END_STRUCT;
      TON_OP_REST_MissingCnd { S7_SetPoint := 'True'} : TON_TIME;
      TON_OP_WORK_MissingCnd { S7_SetPoint := 'True'} : TON_TIME;
   END_VAR
   VAR_TEMP
      PE : Struct
         OP_Rest_PB : Bool;
         OP_Work_PB : Bool;
      END_STRUCT;
   END_VAR
   VAR_TEMP   // added for the SCL form of the ladder/FBD networks
      _w1 : Bool;
      _w2 : Bool;
      _w3 : Bool;
   END_VAR
BEGIN

REGION Network 2: Operazione può muoversi liberamente perchè non sposta nessun BEAM
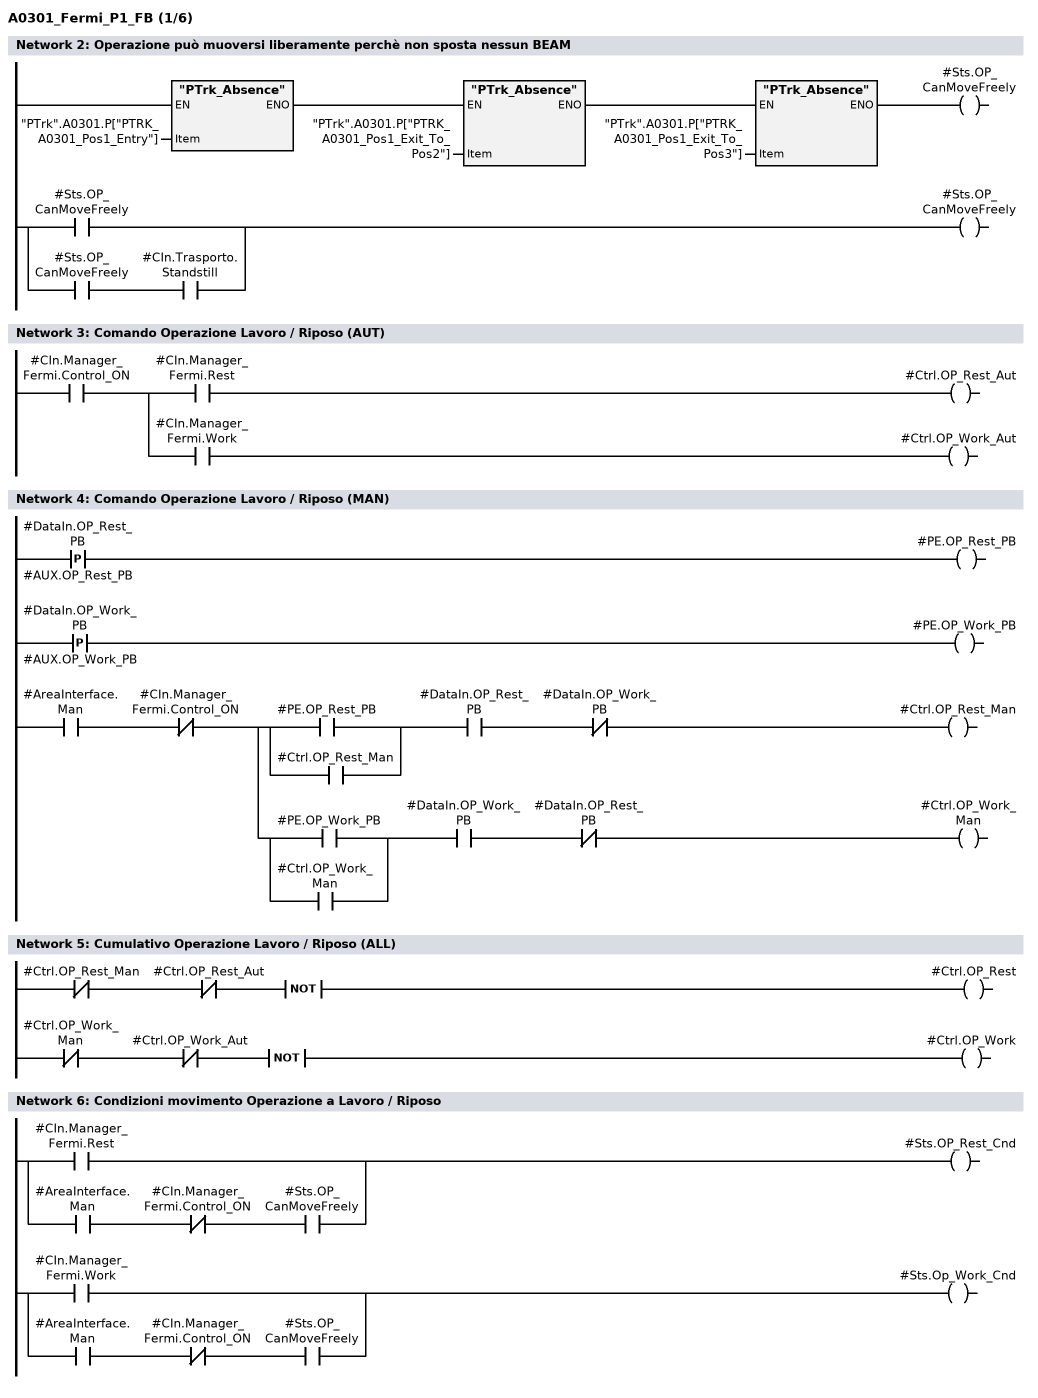
   RUNG wire#powerrail
      "PTrk_Absence"(Item := "PTrk".A0301.P["PTRK_A0301_Pos1_Entry"])
      "PTrk_Absence"(Item := "PTrk".A0301.P["PTRK_A0301_Pos1_Exit_To_Pos2"])
      "PTrk_Absence"(Item := "PTrk".A0301.P["PTRK_A0301_Pos1_Exit_To_Pos3"])
      Coil( #Sts.OP_CanMoveFreely )
   END_RUNG
   RUNG wire#powerrail
      Contact( #Sts.OP_CanMoveFreely )
      wire#w1
      Coil( #Sts.OP_CanMoveFreely )
   END_RUNG
   RUNG wire#powerrail
      Contact( #Sts.OP_CanMoveFreely )
      Contact( #CIn.Trasporto.Standstill )
   END_RUNG wire#w1
   // the same network as SCL:
   "PTrk_Absence"(Item := "PTrk".A0301.P["PTRK_A0301_Pos1_Entry"], ENO => #_w1);
   "PTrk_Absence"(EN := #_w1, Item := "PTrk".A0301.P["PTRK_A0301_Pos1_Exit_To_Pos2"], ENO => #_w2);
   "PTrk_Absence"(EN := #_w2, Item := "PTrk".A0301.P["PTRK_A0301_Pos1_Exit_To_Pos3"], ENO => #_w3);
   #Sts.OP_CanMoveFreely := #_w3;
   #Sts.OP_CanMoveFreely := #Sts.OP_CanMoveFreely OR (#Sts.OP_CanMoveFreely AND #CIn.Trasporto.Standstill);
END_REGION

REGION Network 3: Comando Operazione Lavoro / Riposo (AUT)
   RUNG wire#powerrail
      Contact( #CIn.Manager_Fermi.Control_ON )
      wire#w1
      Contact( #CIn.Manager_Fermi.Rest )
      Coil( #Ctrl.OP_Rest_Aut )
   END_RUNG
   RUNG wire#w1
      Contact( #CIn.Manager_Fermi.Work )
      Coil( #Ctrl.OP_Work_Aut )
   END_RUNG
   // the same network as SCL:
   #Ctrl.OP_Rest_Aut := #CIn.Manager_Fermi.Control_ON AND #CIn.Manager_Fermi.Rest;
   #Ctrl.OP_Work_Aut := #CIn.Manager_Fermi.Control_ON AND #CIn.Manager_Fermi.Work;
END_REGION

REGION Network 4: Comando Operazione Lavoro / Riposo (MAN)
   RUNG wire#powerrail
      P_Contact(operand := #DataIn.OP_Rest_PB, bit := #AUX.OP_Rest_PB)
      Coil( #PE.OP_Rest_PB )
   END_RUNG
   RUNG wire#powerrail
      P_Contact(operand := #DataIn.OP_Work_PB, bit := #AUX.OP_Work_PB)
      Coil( #PE.OP_Work_PB )
   END_RUNG
   RUNG wire#powerrail
      Contact( #AreaInterface.Man )
      I_Contact( #CIn.Manager_Fermi.Control_ON )
      wire#w1
      Contact( #PE.OP_Rest_PB )
      wire#w2
      Contact( #DataIn.OP_Rest_PB )
      I_Contact( #DataIn.OP_Work_PB )
      Coil( #Ctrl.OP_Rest_Man )
   END_RUNG
   RUNG wire#w1
      Contact( #Ctrl.OP_Rest_Man )
   END_RUNG wire#w2
   RUNG wire#w1
      Contact( #PE.OP_Work_PB )
      wire#w3
      Contact( #DataIn.OP_Work_PB )
      I_Contact( #DataIn.OP_Rest_PB )
      Coil( #Ctrl.OP_Work_Man )
   END_RUNG
   RUNG wire#w1
      Contact( #Ctrl.OP_Work_Man )
   END_RUNG wire#w3
   // the same network as SCL:
   #_w1 := #DataIn.OP_Rest_PB AND NOT #AUX.OP_Rest_PB;   // rising edge of #DataIn.OP_Rest_PB
   #AUX.OP_Rest_PB := #DataIn.OP_Rest_PB;
   #PE.OP_Rest_PB := #_w1;
   #_w2 := #DataIn.OP_Work_PB AND NOT #AUX.OP_Work_PB;   // rising edge of #DataIn.OP_Work_PB
   #AUX.OP_Work_PB := #DataIn.OP_Work_PB;
   #PE.OP_Work_PB := #_w2;
   #_w3 := #AreaInterface.Man AND NOT #CIn.Manager_Fermi.Control_ON;
   #Ctrl.OP_Rest_Man := #_w3 AND (#PE.OP_Rest_PB OR #Ctrl.OP_Rest_Man) AND #DataIn.OP_Rest_PB AND NOT #DataIn.OP_Work_PB;
   #Ctrl.OP_Work_Man := #_w3 AND (#PE.OP_Work_PB OR #Ctrl.OP_Work_Man) AND #DataIn.OP_Work_PB AND NOT #DataIn.OP_Rest_PB;
END_REGION

REGION Network 5: Cumulativo Operazione Lavoro / Riposo (ALL)
   RUNG wire#powerrail
      I_Contact( #Ctrl.OP_Rest_Man )
      I_Contact( #Ctrl.OP_Rest_Aut )
      Not()
      Coil( #Ctrl.OP_Rest )
   END_RUNG
   RUNG wire#powerrail
      I_Contact( #Ctrl.OP_Work_Man )
      I_Contact( #Ctrl.OP_Work_Aut )
      Not()
      Coil( #Ctrl.OP_Work )
   END_RUNG
   // the same network as SCL:
   #Ctrl.OP_Rest := NOT (NOT #Ctrl.OP_Rest_Man AND NOT #Ctrl.OP_Rest_Aut);
   #Ctrl.OP_Work := NOT (NOT #Ctrl.OP_Work_Man AND NOT #Ctrl.OP_Work_Aut);
END_REGION

REGION Network 6: Condizioni movimento Operazione a Lavoro / Riposo
   RUNG wire#powerrail
      Contact( #CIn.Manager_Fermi.Rest )
      wire#w1
      Coil( #Sts.OP_Rest_Cnd )
   END_RUNG
   RUNG wire#powerrail
      Contact( #AreaInterface.Man )
      I_Contact( #CIn.Manager_Fermi.Control_ON )
      Contact( #Sts.OP_CanMoveFreely )
   END_RUNG wire#w1
   RUNG wire#powerrail
      Contact( #CIn.Manager_Fermi.Work )
      wire#w2
      Coil( #Sts.Op_Work_Cnd )
   END_RUNG
   RUNG wire#powerrail
      Contact( #AreaInterface.Man )
      I_Contact( #CIn.Manager_Fermi.Control_ON )
      Contact( #Sts.OP_CanMoveFreely )
   END_RUNG wire#w2
   // the same network as SCL:
   #Sts.OP_Rest_Cnd := #CIn.Manager_Fermi.Rest OR (#AreaInterface.Man AND NOT #CIn.Manager_Fermi.Control_ON AND #Sts.OP_CanMoveFreely);
   #Sts.Op_Work_Cnd := #CIn.Manager_Fermi.Work OR (#AreaInterface.Man AND NOT #CIn.Manager_Fermi.Control_ON AND #Sts.OP_CanMoveFreely);
END_REGION

REGION Network 8 (SCL): Fermi + Pareggiatore + Sfalsatore - Cin Manager (Esecuzione sequenza comandi)
   //
   #Fermi[1].Cin.Manager.Rest := FALSE;
   #Fermi[2].Cin.Manager.Rest := FALSE;
   #Fermi[3].Cin.Manager.Rest := FALSE;
   #Fermi[4].Cin.Manager.Rest := FALSE;
   #Fermi[5].Cin.Manager.Rest := FALSE;
   #Fermi[6].Cin.Manager.Rest := FALSE;
   //************************************
   #Fermi[1].Cin.Manager.Work := FALSE;
   #Fermi[2].Cin.Manager.Work := FALSE;
   #Fermi[3].Cin.Manager.Work := FALSE;
   #Fermi[4].Cin.Manager.Work := FALSE;
   #Fermi[5].Cin.Manager.Work := FALSE;
   #Fermi[6].Cin.Manager.Work := FALSE;
   #Pareggiatore.Cin.Manager.Work := FALSE;
   //
   // CIn Manager  Control ON se ho un richiesta di comando attiva
   IF #AreaInterface.Aut OR #CIn.SemiAut THEN
       #Fermi[1].Cin.Manager.Control_ON := TRUE;
       #Fermi[2].Cin.Manager.Control_ON := TRUE;
       #Fermi[3].Cin.Manager.Control_ON := TRUE;
       #Fermi[4].Cin.Manager.Control_ON := TRUE;
       #Fermi[5].Cin.Manager.Control_ON := TRUE;
       #Fermi[6].Cin.Manager.Control_ON := TRUE;
   ELSE
       #Fermi[1].Cin.Manager.Control_ON := FALSE;
       #Fermi[2].Cin.Manager.Control_ON := FALSE;
       #Fermi[3].Cin.Manager.Control_ON := FALSE;
       #Fermi[4].Cin.Manager.Control_ON := FALSE;
       #Fermi[5].Cin.Manager.Control_ON := FALSE;
       #Fermi[6].Cin.Manager.Control_ON := FALSE;
   END_IF;

   // Comando CIn Manager Work FERMI se Sfalsatore indietro
   IF #Ctrl.OP_Work AND #Sts.Op_Work_Cnd THEN

       #Fermi[1].Cin.Manager.Work := TRUE;
       #Fermi[2].Cin.Manager.Work := TRUE;
       #Fermi[3].Cin.Manager.Work := TRUE;
       #Fermi[4].Cin.Manager.Work := TRUE;
       #Fermi[5].Cin.Manager.Work := TRUE;
       #Fermi[6].Cin.Manager.Work := TRUE;

   END_IF;


   // Comando CIn Manager Rest FERMI se Sfalsatore è basso
   IF #Ctrl.OP_Rest AND #Sts.OP_Rest_Cnd THEN

   #Fermi[1].Cin.Manager.Rest := TRUE;
   #Fermi[2].Cin.Manager.Rest := TRUE;
   #Fermi[3].Cin.Manager.Rest := TRUE;
   #Fermi[4].Cin.Manager.Rest := TRUE;
   #Fermi[5].Cin.Manager.Rest := TRUE;
   #Fermi[6].Cin.Manager.Rest := TRUE;

   END_IF;
END_REGION

REGION Network 9 (SCL): CIn Abilitazioni Stop Manager
   //
   // CIn Manager Stop per richiesta apertura safety
   IF #CIn.Manager_Fermi.EnableStopDoorOpeningReq THEN
       #Fermi[1].Cin.Manager.EnableStopDoorOpeningReq := TRUE;
       #Fermi[2].Cin.Manager.EnableStopDoorOpeningReq := TRUE;
       #Fermi[3].Cin.Manager.EnableStopDoorOpeningReq := TRUE;
       #Fermi[4].Cin.Manager.EnableStopDoorOpeningReq := TRUE;
       #Fermi[5].Cin.Manager.EnableStopDoorOpeningReq := TRUE;
       #Fermi[6].Cin.Manager.EnableStopDoorOpeningReq := TRUE;
       #Pareggiatore.Cin.Manager.EnableStopDoorOpeningReq := TRUE;
   ELSE
       #Fermi[1].Cin.Manager.EnableStopDoorOpeningReq := FALSE;
       #Fermi[2].Cin.Manager.EnableStopDoorOpeningReq := FALSE;
       #Fermi[3].Cin.Manager.EnableStopDoorOpeningReq := FALSE;
       #Fermi[4].Cin.Manager.EnableStopDoorOpeningReq := FALSE;
       #Fermi[5].Cin.Manager.EnableStopDoorOpeningReq := FALSE;
       #Fermi[6].Cin.Manager.EnableStopDoorOpeningReq := FALSE;
       #Pareggiatore.Cin.Manager.EnableStopDoorOpeningReq := FALSE;
   END_IF;
   // CIn Manager Stop in fase delle macchine precedenti
   IF #CIn.Manager_Fermi.EnableStopInPhase THEN
       #Fermi[1].Cin.Manager.EnableStopInPhase := TRUE;
       #Fermi[2].Cin.Manager.EnableStopInPhase := TRUE;
       #Fermi[3].Cin.Manager.EnableStopInPhase := TRUE;
       #Fermi[4].Cin.Manager.EnableStopInPhase := TRUE;
       #Fermi[5].Cin.Manager.EnableStopInPhase := TRUE;
       #Fermi[6].Cin.Manager.EnableStopInPhase := TRUE;
       #Pareggiatore.Cin.Manager.EnableStopInPhase := TRUE;
   ELSE
       #Fermi[1].Cin.Manager.EnableStopInPhase := FALSE;
       #Fermi[2].Cin.Manager.EnableStopInPhase := FALSE;
       #Fermi[3].Cin.Manager.EnableStopInPhase := FALSE;
       #Fermi[4].Cin.Manager.EnableStopInPhase := FALSE;
       #Fermi[5].Cin.Manager.EnableStopInPhase := FALSE;
       #Fermi[6].Cin.Manager.EnableStopInPhase := FALSE;
       #Pareggiatore.Cin.Manager.EnableStopInPhase := FALSE;
   END_IF;

   // CIn Manager Stop programmato configurabile a piacere
   IF #CIn.Manager_Fermi.EnableStopProgrammed THEN
       #Fermi[1].Cin.Manager.EnableStopProgrammed := TRUE;
       #Fermi[2].Cin.Manager.EnableStopProgrammed := TRUE;
       #Fermi[3].Cin.Manager.EnableStopProgrammed := TRUE;
       #Fermi[4].Cin.Manager.EnableStopProgrammed := TRUE;
       #Fermi[5].Cin.Manager.EnableStopProgrammed := TRUE;
       #Fermi[6].Cin.Manager.EnableStopProgrammed := TRUE;
       #Pareggiatore.Cin.Manager.EnableStopProgrammed := TRUE;
   ELSE
       #Fermi[1].Cin.Manager.EnableStopProgrammed := FALSE;
       #Fermi[2].Cin.Manager.EnableStopProgrammed := FALSE;
       #Fermi[3].Cin.Manager.EnableStopProgrammed := FALSE;
       #Fermi[4].Cin.Manager.EnableStopProgrammed := FALSE;
       #Fermi[5].Cin.Manager.EnableStopProgrammed := FALSE;
       #Fermi[6].Cin.Manager.EnableStopProgrammed := FALSE;
       #Pareggiatore.Cin.Manager.EnableStopProgrammed := FALSE;
   END_IF;
END_REGION

REGION Network 10: <+>
END_REGION

REGION Network 11: Warning manacanza condizioni esecuzione Operazione RIPOSO / LAVORO
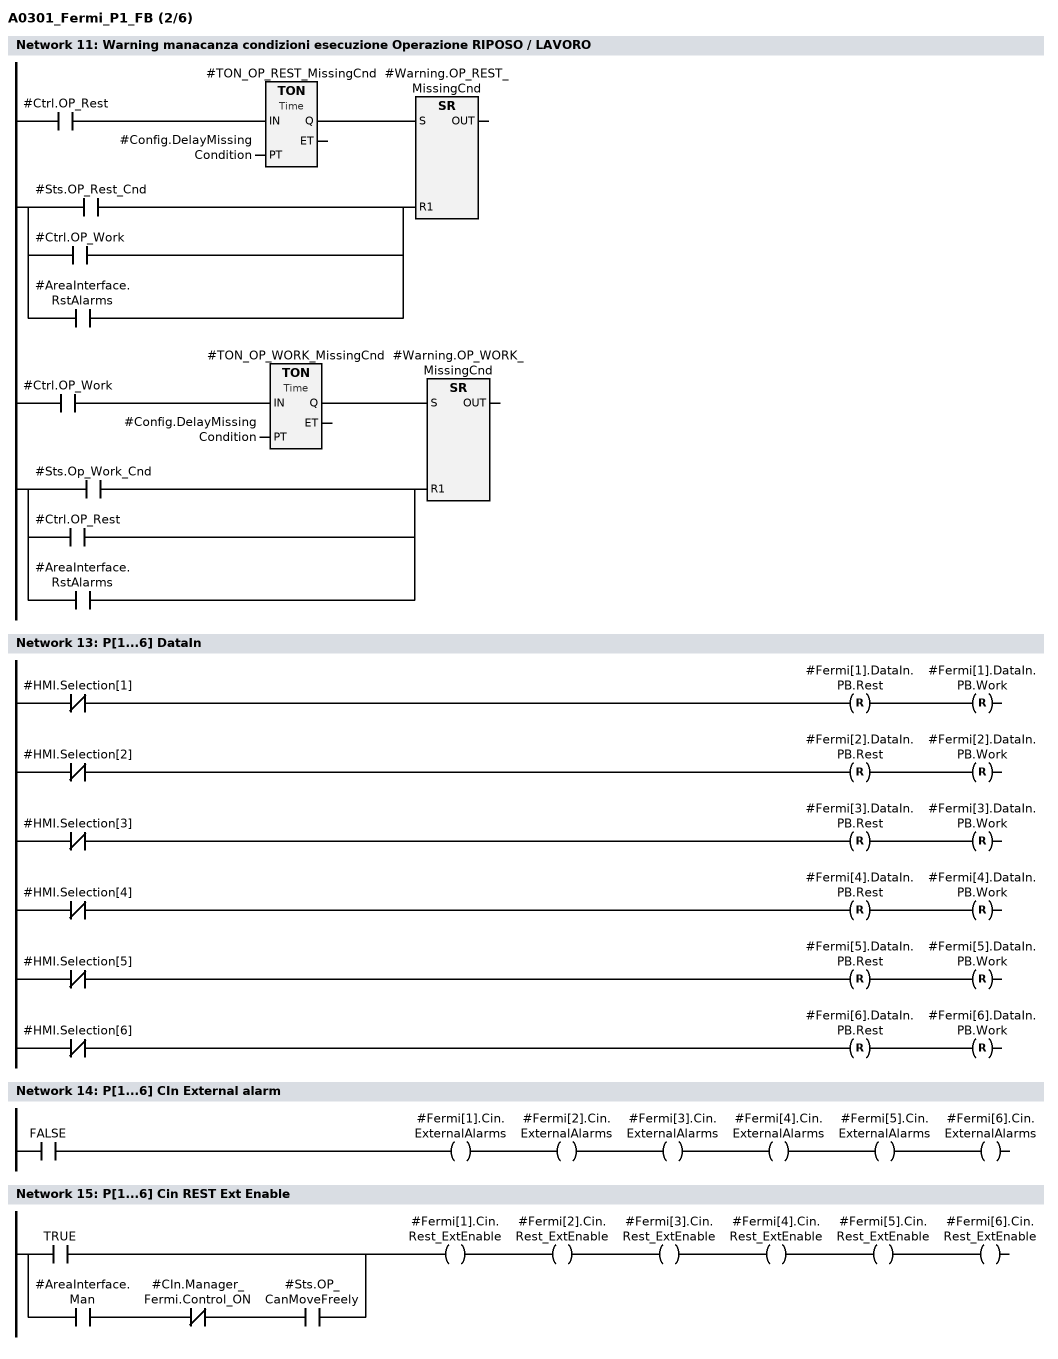
   RUNG wire#powerrail
      Contact( #Ctrl.OP_Rest )
      { S7_Templates := "time_type := Time" } #TON_OP_REST_MissingCnd.TON(pt := #Config.DelayMissingCondition, et =>)
      S_SR(operand := #Warning.OP_REST_MissingCnd, r1 := wire#w1)
   END_RUNG
   RUNG wire#powerrail
      Contact( #Sts.OP_Rest_Cnd )
   END_RUNG wire#w1
   RUNG wire#powerrail
      Contact( #Ctrl.OP_Work )
   END_RUNG wire#w1
   RUNG wire#powerrail
      Contact( #AreaInterface.RstAlarms )
   END_RUNG wire#w1
   RUNG wire#powerrail
      Contact( #Ctrl.OP_Work )
      { S7_Templates := "time_type := Time" } #TON_OP_WORK_MissingCnd.TON(pt := #Config.DelayMissingCondition, et =>)
      S_SR(operand := #Warning.OP_WORK_MissingCnd, r1 := wire#w2)
   END_RUNG
   RUNG wire#powerrail
      Contact( #Sts.Op_Work_Cnd )
   END_RUNG wire#w2
   RUNG wire#powerrail
      Contact( #Ctrl.OP_Rest )
   END_RUNG wire#w2
   RUNG wire#powerrail
      Contact( #AreaInterface.RstAlarms )
   END_RUNG wire#w2
   // the same network as SCL:
   #TON_OP_REST_MissingCnd(IN := #Ctrl.OP_Rest, PT := #Config.DelayMissingCondition);   // TON
   IF #TON_OP_REST_MissingCnd.Q THEN
       #Warning.OP_REST_MissingCnd := TRUE;   // SR flip-flop
   END_IF;
   IF #Sts.OP_Rest_Cnd OR #Ctrl.OP_Work OR #AreaInterface.RstAlarms THEN
       #Warning.OP_REST_MissingCnd := FALSE;
   END_IF;
   #TON_OP_WORK_MissingCnd(IN := #Ctrl.OP_Work, PT := #Config.DelayMissingCondition);   // TON
   IF #TON_OP_WORK_MissingCnd.Q THEN
       #Warning.OP_WORK_MissingCnd := TRUE;   // SR flip-flop
   END_IF;
   IF #Sts.Op_Work_Cnd OR #Ctrl.OP_Rest OR #AreaInterface.RstAlarms THEN
       #Warning.OP_WORK_MissingCnd := FALSE;
   END_IF;
END_REGION

REGION Network 12: << GESTIONE FERMI >>
END_REGION

REGION Network 13: P[1...6] DataIn
   RUNG wire#powerrail
      I_Contact( #HMI.Selection[1] )
      R_Coil( #Fermi[1].DataIn.PB.Rest )
      R_Coil( #Fermi[1].DataIn.PB.Work )
   END_RUNG
   RUNG wire#powerrail
      I_Contact( #HMI.Selection[2] )
      R_Coil( #Fermi[2].DataIn.PB.Rest )
      R_Coil( #Fermi[2].DataIn.PB.Work )
   END_RUNG
   RUNG wire#powerrail
      I_Contact( #HMI.Selection[3] )
      R_Coil( #Fermi[3].DataIn.PB.Rest )
      R_Coil( #Fermi[3].DataIn.PB.Work )
   END_RUNG
   RUNG wire#powerrail
      I_Contact( #HMI.Selection[4] )
      R_Coil( #Fermi[4].DataIn.PB.Rest )
      R_Coil( #Fermi[4].DataIn.PB.Work )
   END_RUNG
   RUNG wire#powerrail
      I_Contact( #HMI.Selection[5] )
      R_Coil( #Fermi[5].DataIn.PB.Rest )
      R_Coil( #Fermi[5].DataIn.PB.Work )
   END_RUNG
   RUNG wire#powerrail
      I_Contact( #HMI.Selection[6] )
      R_Coil( #Fermi[6].DataIn.PB.Rest )
      R_Coil( #Fermi[6].DataIn.PB.Work )
   END_RUNG
   // the same network as SCL:
   IF NOT #HMI.Selection[1] THEN
       #Fermi[1].DataIn.PB.Rest := FALSE;
       #Fermi[1].DataIn.PB.Work := FALSE;
   END_IF;
   IF NOT #HMI.Selection[2] THEN
       #Fermi[2].DataIn.PB.Rest := FALSE;
       #Fermi[2].DataIn.PB.Work := FALSE;
   END_IF;
   IF NOT #HMI.Selection[3] THEN
       #Fermi[3].DataIn.PB.Rest := FALSE;
       #Fermi[3].DataIn.PB.Work := FALSE;
   END_IF;
   IF NOT #HMI.Selection[4] THEN
       #Fermi[4].DataIn.PB.Rest := FALSE;
       #Fermi[4].DataIn.PB.Work := FALSE;
   END_IF;
   IF NOT #HMI.Selection[5] THEN
       #Fermi[5].DataIn.PB.Rest := FALSE;
       #Fermi[5].DataIn.PB.Work := FALSE;
   END_IF;
   IF NOT #HMI.Selection[6] THEN
       #Fermi[6].DataIn.PB.Rest := FALSE;
       #Fermi[6].DataIn.PB.Work := FALSE;
   END_IF;
END_REGION

REGION Network 14: P[1...6] CIn External alarm
   RUNG wire#powerrail
      Contact( FALSE )
      Coil( #Fermi[1].Cin.ExternalAlarms )
      Coil( #Fermi[2].Cin.ExternalAlarms )
      Coil( #Fermi[3].Cin.ExternalAlarms )
      Coil( #Fermi[4].Cin.ExternalAlarms )
      Coil( #Fermi[5].Cin.ExternalAlarms )
      Coil( #Fermi[6].Cin.ExternalAlarms )
   END_RUNG
   // the same network as SCL:
   #Fermi[1].Cin.ExternalAlarms := FALSE;
   #Fermi[2].Cin.ExternalAlarms := FALSE;
   #Fermi[3].Cin.ExternalAlarms := FALSE;
   #Fermi[4].Cin.ExternalAlarms := FALSE;
   #Fermi[5].Cin.ExternalAlarms := FALSE;
   #Fermi[6].Cin.ExternalAlarms := FALSE;
END_REGION

REGION Network 15: P[1...6] Cin REST Ext Enable
   RUNG wire#powerrail
      Contact( TRUE )
      wire#w1
      Coil( #Fermi[1].Cin.Rest_ExtEnable )
      Coil( #Fermi[2].Cin.Rest_ExtEnable )
      Coil( #Fermi[3].Cin.Rest_ExtEnable )
      Coil( #Fermi[4].Cin.Rest_ExtEnable )
      Coil( #Fermi[5].Cin.Rest_ExtEnable )
      Coil( #Fermi[6].Cin.Rest_ExtEnable )
   END_RUNG
   RUNG wire#powerrail
      Contact( #AreaInterface.Man )
      I_Contact( #CIn.Manager_Fermi.Control_ON )
      Contact( #Sts.OP_CanMoveFreely )
   END_RUNG wire#w1
   // the same network as SCL:
   #Fermi[1].Cin.Rest_ExtEnable := TRUE OR (#AreaInterface.Man AND NOT #CIn.Manager_Fermi.Control_ON AND #Sts.OP_CanMoveFreely);
   #Fermi[2].Cin.Rest_ExtEnable := TRUE OR (#AreaInterface.Man AND NOT #CIn.Manager_Fermi.Control_ON AND #Sts.OP_CanMoveFreely);
   #Fermi[3].Cin.Rest_ExtEnable := TRUE OR (#AreaInterface.Man AND NOT #CIn.Manager_Fermi.Control_ON AND #Sts.OP_CanMoveFreely);
   #Fermi[4].Cin.Rest_ExtEnable := TRUE OR (#AreaInterface.Man AND NOT #CIn.Manager_Fermi.Control_ON AND #Sts.OP_CanMoveFreely);
   #Fermi[5].Cin.Rest_ExtEnable := TRUE OR (#AreaInterface.Man AND NOT #CIn.Manager_Fermi.Control_ON AND #Sts.OP_CanMoveFreely);
   #Fermi[6].Cin.Rest_ExtEnable := TRUE OR (#AreaInterface.Man AND NOT #CIn.Manager_Fermi.Control_ON AND #Sts.OP_CanMoveFreely);
END_REGION

REGION Network 16: P[1...6] Cin WORK Ext Enable
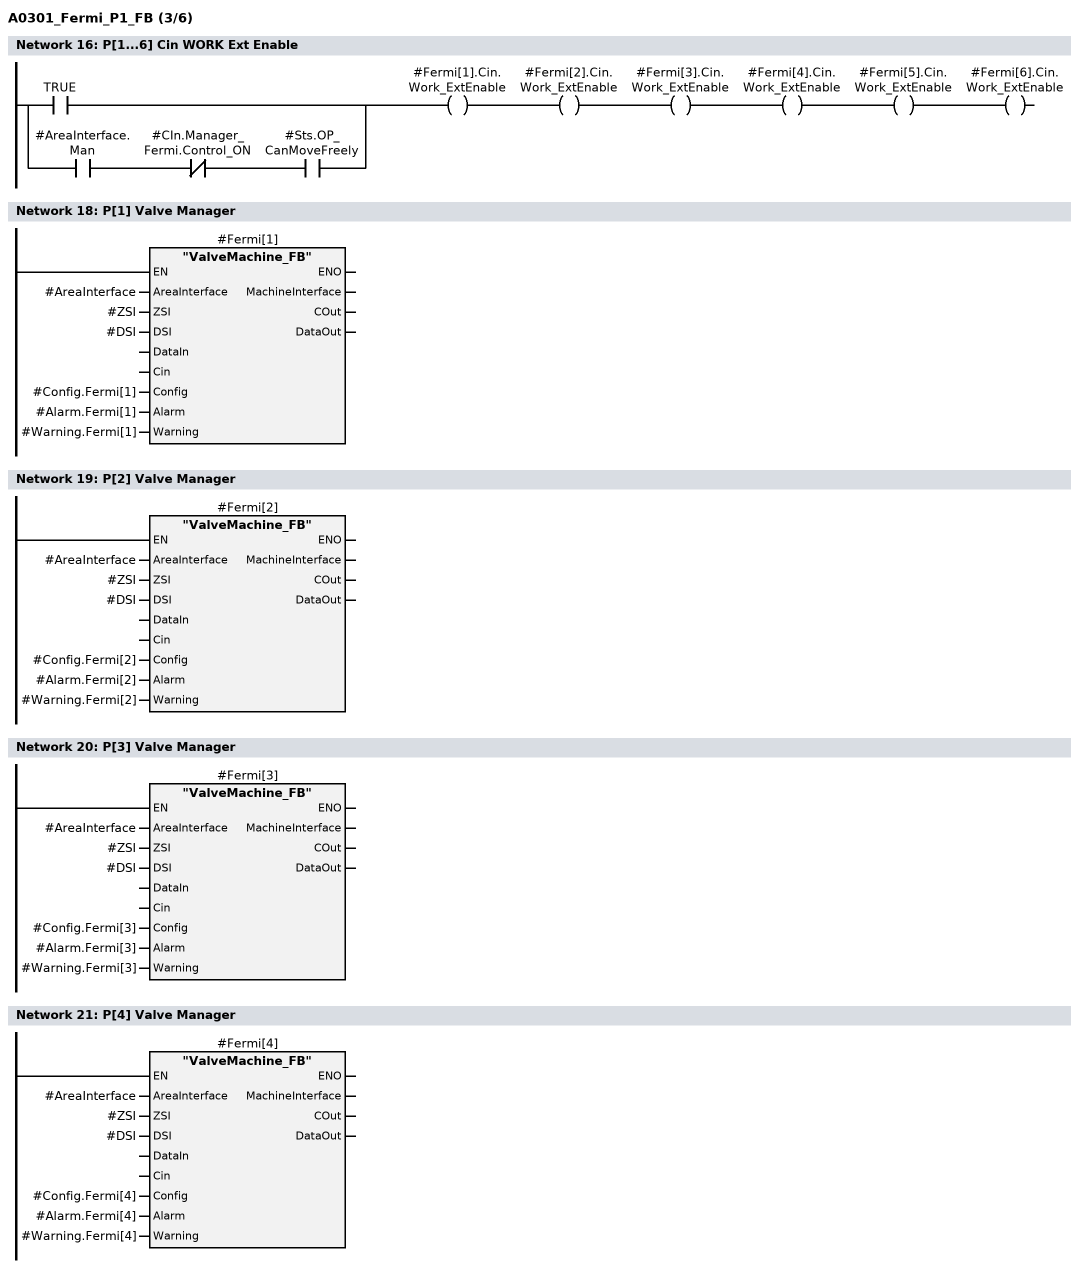
   RUNG wire#powerrail
      Contact( TRUE )
      wire#w1
      Coil( #Fermi[1].Cin.Work_ExtEnable )
      Coil( #Fermi[2].Cin.Work_ExtEnable )
      Coil( #Fermi[3].Cin.Work_ExtEnable )
      Coil( #Fermi[4].Cin.Work_ExtEnable )
      Coil( #Fermi[5].Cin.Work_ExtEnable )
      Coil( #Fermi[6].Cin.Work_ExtEnable )
   END_RUNG
   RUNG wire#powerrail
      Contact( #AreaInterface.Man )
      I_Contact( #CIn.Manager_Fermi.Control_ON )
      Contact( #Sts.OP_CanMoveFreely )
   END_RUNG wire#w1
   // the same network as SCL:
   #Fermi[1].Cin.Work_ExtEnable := TRUE OR (#AreaInterface.Man AND NOT #CIn.Manager_Fermi.Control_ON AND #Sts.OP_CanMoveFreely);
   #Fermi[2].Cin.Work_ExtEnable := TRUE OR (#AreaInterface.Man AND NOT #CIn.Manager_Fermi.Control_ON AND #Sts.OP_CanMoveFreely);
   #Fermi[3].Cin.Work_ExtEnable := TRUE OR (#AreaInterface.Man AND NOT #CIn.Manager_Fermi.Control_ON AND #Sts.OP_CanMoveFreely);
   #Fermi[4].Cin.Work_ExtEnable := TRUE OR (#AreaInterface.Man AND NOT #CIn.Manager_Fermi.Control_ON AND #Sts.OP_CanMoveFreely);
   #Fermi[5].Cin.Work_ExtEnable := TRUE OR (#AreaInterface.Man AND NOT #CIn.Manager_Fermi.Control_ON AND #Sts.OP_CanMoveFreely);
   #Fermi[6].Cin.Work_ExtEnable := TRUE OR (#AreaInterface.Man AND NOT #CIn.Manager_Fermi.Control_ON AND #Sts.OP_CanMoveFreely);
END_REGION

REGION Network 17: <+>
END_REGION

REGION Network 18: P[1] Valve Manager
   RUNG wire#powerrail
      #Fermi[1](AreaInterface := #AreaInterface, ZSI := #ZSI, DSI := #DSI, DataIn :=, Cin :=, Config := #Config.Fermi[1], Alarm := #Alarm.Fermi[1], Warning := #Warning.Fermi[1], MachineInterface =>, COut =>, DataOut =>)
   END_RUNG
   // the same network as SCL:
   #Fermi[1](AreaInterface := #AreaInterface,   // "ValveMachine_FB"
             ZSI := #ZSI,
             DSI := #DSI,
             Config := #Config.Fermi[1],
             Alarm := #Alarm.Fermi[1],
             Warning := #Warning.Fermi[1]);
END_REGION

REGION Network 19: P[2] Valve Manager
   RUNG wire#powerrail
      #Fermi[2](AreaInterface := #AreaInterface, ZSI := #ZSI, DSI := #DSI, DataIn :=, Cin :=, Config := #Config.Fermi[2], Alarm := #Alarm.Fermi[2], Warning := #Warning.Fermi[2], MachineInterface =>, COut =>, DataOut =>)
   END_RUNG
   // the same network as SCL:
   #Fermi[2](AreaInterface := #AreaInterface,   // "ValveMachine_FB"
             ZSI := #ZSI,
             DSI := #DSI,
             Config := #Config.Fermi[2],
             Alarm := #Alarm.Fermi[2],
             Warning := #Warning.Fermi[2]);
END_REGION

REGION Network 20: P[3] Valve Manager
   RUNG wire#powerrail
      #Fermi[3](AreaInterface := #AreaInterface, ZSI := #ZSI, DSI := #DSI, DataIn :=, Cin :=, Config := #Config.Fermi[3], Alarm := #Alarm.Fermi[3], Warning := #Warning.Fermi[3], MachineInterface =>, COut =>, DataOut =>)
   END_RUNG
   // the same network as SCL:
   #Fermi[3](AreaInterface := #AreaInterface,   // "ValveMachine_FB"
             ZSI := #ZSI,
             DSI := #DSI,
             Config := #Config.Fermi[3],
             Alarm := #Alarm.Fermi[3],
             Warning := #Warning.Fermi[3]);
END_REGION

REGION Network 21: P[4] Valve Manager
   RUNG wire#powerrail
      #Fermi[4](AreaInterface := #AreaInterface, ZSI := #ZSI, DSI := #DSI, DataIn :=, Cin :=, Config := #Config.Fermi[4], Alarm := #Alarm.Fermi[4], Warning := #Warning.Fermi[4], MachineInterface =>, COut =>, DataOut =>)
   END_RUNG
   // the same network as SCL:
   #Fermi[4](AreaInterface := #AreaInterface,   // "ValveMachine_FB"
             ZSI := #ZSI,
             DSI := #DSI,
             Config := #Config.Fermi[4],
             Alarm := #Alarm.Fermi[4],
             Warning := #Warning.Fermi[4]);
END_REGION

REGION Network 22: P[5] Valve Manager
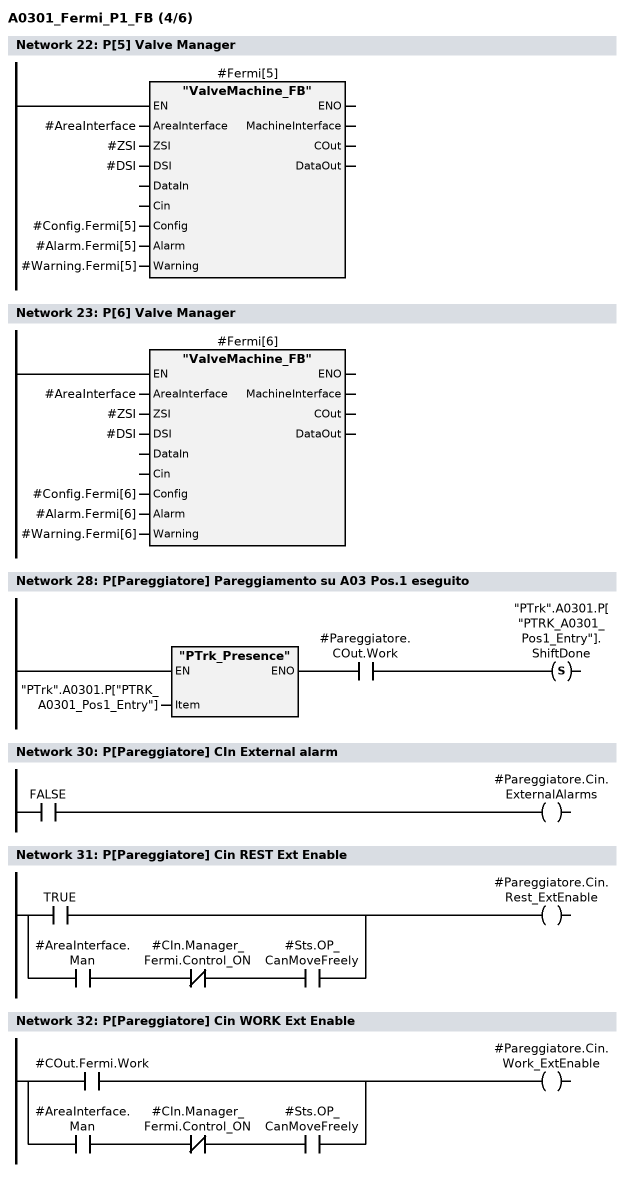
   RUNG wire#powerrail
      #Fermi[5](AreaInterface := #AreaInterface, ZSI := #ZSI, DSI := #DSI, DataIn :=, Cin :=, Config := #Config.Fermi[5], Alarm := #Alarm.Fermi[5], Warning := #Warning.Fermi[5], MachineInterface =>, COut =>, DataOut =>)
   END_RUNG
   // the same network as SCL:
   #Fermi[5](AreaInterface := #AreaInterface,   // "ValveMachine_FB"
             ZSI := #ZSI,
             DSI := #DSI,
             Config := #Config.Fermi[5],
             Alarm := #Alarm.Fermi[5],
             Warning := #Warning.Fermi[5]);
END_REGION

REGION Network 23: P[6] Valve Manager
   RUNG wire#powerrail
      #Fermi[6](AreaInterface := #AreaInterface, ZSI := #ZSI, DSI := #DSI, DataIn :=, Cin :=, Config := #Config.Fermi[6], Alarm := #Alarm.Fermi[6], Warning := #Warning.Fermi[6], MachineInterface =>, COut =>, DataOut =>)
   END_RUNG
   // the same network as SCL:
   #Fermi[6](AreaInterface := #AreaInterface,   // "ValveMachine_FB"
             ZSI := #ZSI,
             DSI := #DSI,
             Config := #Config.Fermi[6],
             Alarm := #Alarm.Fermi[6],
             Warning := #Warning.Fermi[6]);
END_REGION

REGION Network 24: <+>
END_REGION

REGION Network 25 (SCL): P[1...6] COut Fermi
   REGION COut STANDSTILL Fermi
       // Controllo uscita COut STANDSTILL in base allo stato di tutti i Pin
       IF #Fermi[1].Sts.Standstill AND
          #Fermi[2].Sts.Standstill AND
          #Fermi[3].Sts.Standstill AND
          #Fermi[4].Sts.Standstill AND
          #Fermi[5].Sts.Standstill AND
          #Fermi[6].Sts.Standstill THEN
           #COut.Fermi.Standstill := TRUE;
       ELSE
           #COut.Fermi.Standstill := FALSE;
       END_IF;
   END_REGION ;


   REGION COut AT REST #Fermi
       // Controllo uscita COut AT_REST in base allo stato di tutti i Pin
       IF  #Fermi[1].COut.Rest OR #Fermi[1].DataIn.Rest_Ls[1] AND
           #Fermi[2].COut.Rest OR #Fermi[2].DataIn.Rest_Ls[1] AND
           #Fermi[3].COut.Rest OR #Fermi[3].DataIn.Rest_Ls[1] AND
           #Fermi[4].COut.Rest OR #Fermi[4].DataIn.Rest_Ls[1] AND
           #Fermi[5].COut.Rest OR #Fermi[5].DataIn.Rest_Ls[1] AND
           #Fermi[6].COut.Rest OR #Fermi[6].DataIn.Rest_Ls[1] THEN
           #COut.Fermi.Rest := 1;
       ELSE
           #COut.Fermi.Rest := 0;
       END_IF;
   END_REGION ;

   REGION COut AT WORK Fermi
       // Controllo uscita COut AT_WORK in base allo stato di tutti i Pin
       IF #Fermi[1].COut.Work  AND
           #Fermi[2].COut.Work AND
           #Fermi[3].COut.Work AND
           #Fermi[4].COut.Work AND
           #Fermi[5].COut.Work AND
           #Fermi[6].COut.Work THEN
           #COut.Fermi.Work := 1;
       ELSE
           #COut.Fermi.Work := 0;
       END_IF;
   END_REGION ;
END_REGION

REGION Network 27: <<<< GESTIONE PAREGGIATORE - SemiGuscio >>>
END_REGION

REGION Network 28: P[Pareggiatore] Pareggiamento su A03 Pos.1 eseguito
   RUNG wire#powerrail
      "PTrk_Presence"(Item := "PTrk".A0301.P["PTRK_A0301_Pos1_Entry"])
      Contact( #Pareggiatore.COut.Work )
      S_Coil( "PTrk".A0301.P["PTRK_A0301_Pos1_Entry"].ShiftDone )
   END_RUNG
   // the same network as SCL:
   "PTrk_Presence"(Item := "PTrk".A0301.P["PTRK_A0301_Pos1_Entry"], ENO => #_w1);
   IF #_w1 AND #Pareggiatore.COut.Work THEN
       "PTrk".A0301.P["PTRK_A0301_Pos1_Entry"].ShiftDone := TRUE;
   END_IF;
END_REGION

REGION Network 29: <+>
END_REGION

REGION Network 30: P[Pareggiatore] CIn External alarm
   RUNG wire#powerrail
      Contact( FALSE )
      Coil( #Pareggiatore.Cin.ExternalAlarms )
   END_RUNG
   // the same network as SCL:
   #Pareggiatore.Cin.ExternalAlarms := FALSE;
END_REGION

REGION Network 31: P[Pareggiatore] Cin REST Ext Enable
   RUNG wire#powerrail
      Contact( TRUE )
      wire#w1
      Coil( #Pareggiatore.Cin.Rest_ExtEnable )
   END_RUNG
   RUNG wire#powerrail
      Contact( #AreaInterface.Man )
      I_Contact( #CIn.Manager_Fermi.Control_ON )
      Contact( #Sts.OP_CanMoveFreely )
   END_RUNG wire#w1
   // the same network as SCL:
   #Pareggiatore.Cin.Rest_ExtEnable := TRUE OR (#AreaInterface.Man AND NOT #CIn.Manager_Fermi.Control_ON AND #Sts.OP_CanMoveFreely);
END_REGION

REGION Network 32: P[Pareggiatore] Cin WORK Ext Enable
   RUNG wire#powerrail
      Contact( #COut.Fermi.Work )
      wire#w1
      Coil( #Pareggiatore.Cin.Work_ExtEnable )
   END_RUNG
   RUNG wire#powerrail
      Contact( #AreaInterface.Man )
      I_Contact( #CIn.Manager_Fermi.Control_ON )
      Contact( #Sts.OP_CanMoveFreely )
   END_RUNG wire#w1
   // the same network as SCL:
   #Pareggiatore.Cin.Work_ExtEnable := #COut.Fermi.Work OR (#AreaInterface.Man AND NOT #CIn.Manager_Fermi.Control_ON AND #Sts.OP_CanMoveFreely);
END_REGION

REGION Network 33: <+>
END_REGION

REGION Network 34: P[Pareggiatore] Valve Manager
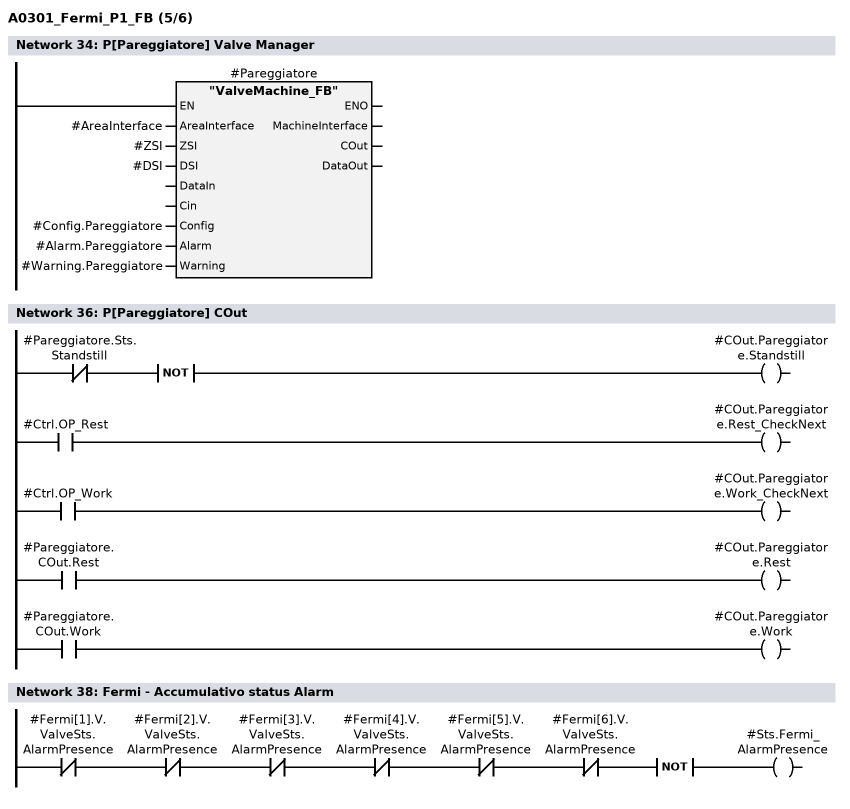
   RUNG wire#powerrail
      #Pareggiatore(AreaInterface := #AreaInterface, ZSI := #ZSI, DSI := #DSI, DataIn :=, Cin :=, Config := #Config.Pareggiatore, Alarm := #Alarm.Pareggiatore, Warning := #Warning.Pareggiatore, MachineInterface =>, COut =>, DataOut =>)
   END_RUNG
   // the same network as SCL:
   #Pareggiatore(AreaInterface := #AreaInterface,   // "ValveMachine_FB"
                 ZSI := #ZSI,
                 DSI := #DSI,
                 Config := #Config.Pareggiatore,
                 Alarm := #Alarm.Pareggiatore,
                 Warning := #Warning.Pareggiatore);
END_REGION

REGION Network 35: <+>
END_REGION

REGION Network 36: P[Pareggiatore] COut
   RUNG wire#powerrail
      I_Contact( #Pareggiatore.Sts.Standstill )
      Not()
      Coil( #COut.Pareggiatore.Standstill )
   END_RUNG
   RUNG wire#powerrail
      Contact( #Ctrl.OP_Rest )
      Coil( #COut.Pareggiatore.Rest_CheckNext )
   END_RUNG
   RUNG wire#powerrail
      Contact( #Ctrl.OP_Work )
      Coil( #COut.Pareggiatore.Work_CheckNext )
   END_RUNG
   RUNG wire#powerrail
      Contact( #Pareggiatore.COut.Rest )
      Coil( #COut.Pareggiatore.Rest )
   END_RUNG
   RUNG wire#powerrail
      Contact( #Pareggiatore.COut.Work )
      Coil( #COut.Pareggiatore.Work )
   END_RUNG
   // the same network as SCL:
   #COut.Pareggiatore.Standstill := NOT (NOT #Pareggiatore.Sts.Standstill);
   #COut.Pareggiatore.Rest_CheckNext := #Ctrl.OP_Rest;
   #COut.Pareggiatore.Work_CheckNext := #Ctrl.OP_Work;
   #COut.Pareggiatore.Rest := #Pareggiatore.COut.Rest;
   #COut.Pareggiatore.Work := #Pareggiatore.COut.Work;
END_REGION

REGION Network 37: <+>
END_REGION

REGION Network 38: Fermi - Accumulativo status Alarm
   RUNG wire#powerrail
      I_Contact( #Fermi[1].V.ValveSts.AlarmPresence )
      I_Contact( #Fermi[2].V.ValveSts.AlarmPresence )
      I_Contact( #Fermi[3].V.ValveSts.AlarmPresence )
      I_Contact( #Fermi[4].V.ValveSts.AlarmPresence )
      I_Contact( #Fermi[5].V.ValveSts.AlarmPresence )
      I_Contact( #Fermi[6].V.ValveSts.AlarmPresence )
      Not()
      Coil( #Sts.Fermi_AlarmPresence )
   END_RUNG
   // the same network as SCL:
   #Sts.Fermi_AlarmPresence := NOT (NOT #Fermi[1].V.ValveSts.AlarmPresence AND NOT #Fermi[2].V.ValveSts.AlarmPresence AND NOT #Fermi[3].V.ValveSts.AlarmPresence AND NOT #Fermi[4].V.ValveSts.AlarmPresence AND NOT #Fermi[5].V.ValveSts.AlarmPresence AND NOT #Fermi[6].V.ValveSts.AlarmPresence);
END_REGION

REGION Network 39 (SCL): HMI STATUS - Postazione
   // Area dati appoggio per HMI
   // FERMI POS.1
   #HMI.FermiSts.Standstill := #COut.Fermi.Standstill;
   #HMI.FermiSts.Rest := #COut.Fermi.Rest;
   #HMI.FermiSts.Work := #COut.Fermi.Work;
   #HMI.FermiSts.AlarmPresence := #Sts.Fermi_AlarmPresence;

   // PAREGGIATORE POS.1
   #HMI.PareggiatoreSts.Standstill := #COut.Pareggiatore.Standstill;
   #HMI.PareggiatoreSts.Rest := #COut.Pareggiatore.Rest;
   #HMI.PareggiatoreSts.Work := #COut.Pareggiatore.Work;
   #HMI.PareggiatoreSts.AlarmPresence := #Pareggiatore.V.ValveSts.AlarmPresence;
END_REGION

REGION Network 41: << MAIN MACHINE STATUS >>
END_REGION

REGION Network 42: Machine interface
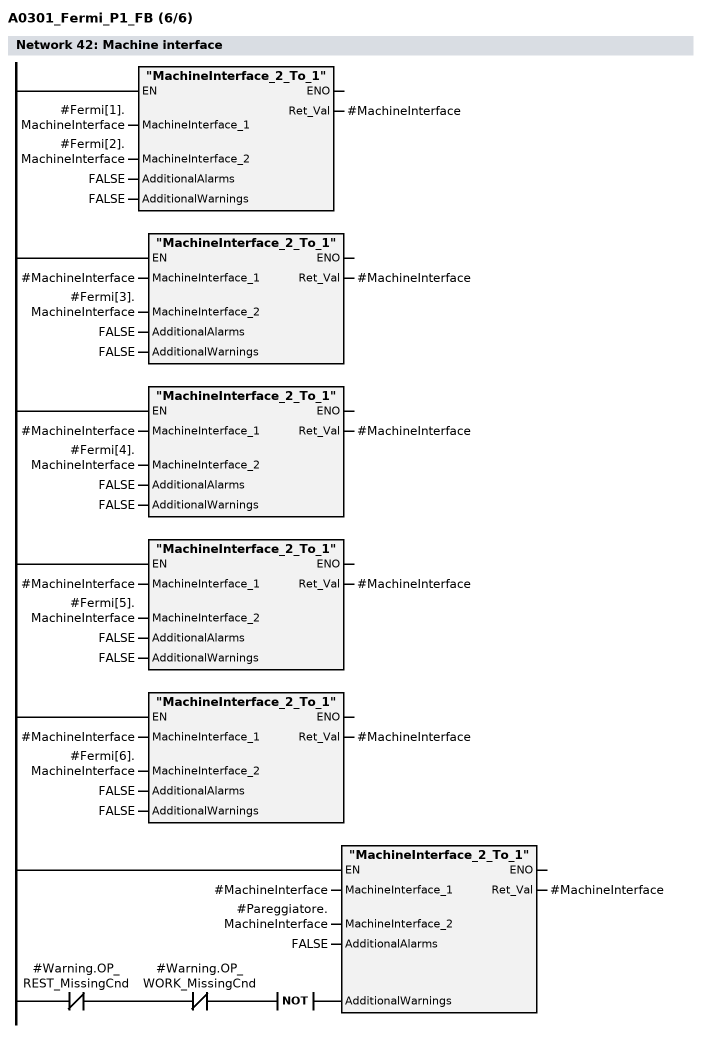
   RUNG wire#powerrail
      "MachineInterface_2_To_1"(MachineInterface_1 := #Fermi[1].MachineInterface, MachineInterface_2 := #Fermi[2].MachineInterface, AdditionalAlarms := FALSE, AdditionalWarnings := FALSE, Ret_Val => #MachineInterface)
   END_RUNG
   RUNG wire#powerrail
      "MachineInterface_2_To_1"(MachineInterface_1 := #MachineInterface, MachineInterface_2 := #Fermi[3].MachineInterface, AdditionalAlarms := FALSE, AdditionalWarnings := FALSE, Ret_Val => #MachineInterface)
   END_RUNG
   RUNG wire#powerrail
      "MachineInterface_2_To_1"(MachineInterface_1 := #MachineInterface, MachineInterface_2 := #Fermi[4].MachineInterface, AdditionalAlarms := FALSE, AdditionalWarnings := FALSE, Ret_Val => #MachineInterface)
   END_RUNG
   RUNG wire#powerrail
      "MachineInterface_2_To_1"(MachineInterface_1 := #MachineInterface, MachineInterface_2 := #Fermi[5].MachineInterface, AdditionalAlarms := FALSE, AdditionalWarnings := FALSE, Ret_Val => #MachineInterface)
   END_RUNG
   RUNG wire#powerrail
      "MachineInterface_2_To_1"(MachineInterface_1 := #MachineInterface, MachineInterface_2 := #Fermi[6].MachineInterface, AdditionalAlarms := FALSE, AdditionalWarnings := FALSE, Ret_Val => #MachineInterface)
   END_RUNG
   RUNG wire#powerrail
      "MachineInterface_2_To_1"(AdditionalWarnings := wire#w1, MachineInterface_1 := #MachineInterface, MachineInterface_2 := #Pareggiatore.MachineInterface, AdditionalAlarms := FALSE, Ret_Val => #MachineInterface)
   END_RUNG
   RUNG wire#powerrail
      I_Contact( #Warning.OP_REST_MissingCnd )
      I_Contact( #Warning.OP_WORK_MissingCnd )
      Not()
   END_RUNG wire#w1
   // the same network as SCL:
   #MachineInterface := "MachineInterface_2_To_1"(MachineInterface_1 := #Fermi[1].MachineInterface,
                           MachineInterface_2 := #Fermi[2].MachineInterface,
                           AdditionalAlarms := FALSE,
                           AdditionalWarnings := FALSE);
   #MachineInterface := "MachineInterface_2_To_1"(MachineInterface_1 := #MachineInterface,
                           MachineInterface_2 := #Fermi[3].MachineInterface,
                           AdditionalAlarms := FALSE,
                           AdditionalWarnings := FALSE);
   #MachineInterface := "MachineInterface_2_To_1"(MachineInterface_1 := #MachineInterface,
                           MachineInterface_2 := #Fermi[4].MachineInterface,
                           AdditionalAlarms := FALSE,
                           AdditionalWarnings := FALSE);
   #MachineInterface := "MachineInterface_2_To_1"(MachineInterface_1 := #MachineInterface,
                           MachineInterface_2 := #Fermi[5].MachineInterface,
                           AdditionalAlarms := FALSE,
                           AdditionalWarnings := FALSE);
   #MachineInterface := "MachineInterface_2_To_1"(MachineInterface_1 := #MachineInterface,
                           MachineInterface_2 := #Fermi[6].MachineInterface,
                           AdditionalAlarms := FALSE,
                           AdditionalWarnings := FALSE);
   #MachineInterface := "MachineInterface_2_To_1"(MachineInterface_1 := #MachineInterface,
                           MachineInterface_2 := #Pareggiatore.MachineInterface,
                           AdditionalAlarms := FALSE,
                           AdditionalWarnings := NOT (NOT #Warning.OP_REST_MissingCnd AND NOT #Warning.OP_WORK_MissingCnd));
END_REGION
END_FUNCTION_BLOCK

FUNCTION "A0301_Fermi_P2_CALL" : Void   // FC86, LAD
// stored: SetENOAutomatically false
BEGIN

REGION Network 1 (SCL): << TRASFERIMENTO stati CIn del blocco >>
   // TRASFERIMENTO #CIn MANAGER
   "A0301_Fermi_P2".CIn.Manager_Fermi := "A0301_Manager".COut.P2.Fermi;
   "A0301_Fermi_P2".CIn.Manager_Sollevatori := "A0301_Manager".COut.P2.Sollevatore;
   //
   "A0301_Fermi_P2".CIn.SemiAut := "A0301_Manager".DataIn.SemiAut_Pb;

   // TRASFERIMENTO #CIn FERMI POSTAZIONI P2 E DEI SOLLEVATORI SU P3
   // Trasferimento status alla Stazione P2 da COut a Cin delle stazioni successive
   "A0301_Fermi_P2".CIn.P1.Fermi := "A0301_Fermi_P1".COut.Fermi;

   // Trasferimento status alla Stazione P2 da COut a Cin dello Sfasatore P1
   "A0301_Fermi_P2".CIn.P1.Pareggiatore := "A0301_Fermi_P1".COut.Pareggiatore;

   REGION TRASFERIMENTO CIn TRASPORTO E RIBALTATORE

       // Trasferimenti status lettura posizioni Ribaltatore al Cin delle stazioni
       "A0301_Fermi_P2".CIn.Sts_Ribalta := "A0301_Ribaltatore".COut.Ribaltatore_Sts;

       // Trasferimenti status lettura posizioni Trasporto al Cin delle stazioni
       "A0301_Fermi_P2".CIn.Trasporto := "A0301_Trasporto".COut.Ax;
   END_REGION ;
END_REGION

REGION Network 2 (SCL): << TRASFERIMENTO stati DataIn >>


   REGION TRASFERIMENTO DataIn DIGITAL INPUT dei LIMIT SWITCH

       // Trasferimento ingressi digitali Limit Switch Fermi P2
       // 
       "A0301_Fermi_P2".Fermi[1].DataIn.Rest_Ls[1] := "A0301_CinghiaTrasporto_1.1_Ls_Rest_7";
       "A0301_Fermi_P2".Fermi[2].DataIn.Rest_Ls[1] := "A0301_CinghiaTrasporto_2.1_Ls_Rest_7";
       "A0301_Fermi_P2".Fermi[3].DataIn.Rest_Ls[1] := "A0301_CinghiaTrasporto_3.1_Ls_Rest_7";
       "A0301_Fermi_P2".Fermi[4].DataIn.Rest_Ls[1] := "A0301_CinghiaTrasporto_4.1_Ls_Rest_7";
       "A0301_Fermi_P2".Fermi[5].DataIn.Rest_Ls[1] := "A0301_CinghiaTrasporto_5.1_Ls_Rest_7";
       "A0301_Fermi_P2".Fermi[6].DataIn.Rest_Ls[1] := "A0301_CinghiaTrasporto_6.1_Ls_Rest_7";

       // Trasferimento ingressi digitali Limit Switch Sollevatori P2
       "A0301_Fermi_P2".Sollevatori[1].DataIn.Rest_Ls[1] := "A0301_CinghiaTrasporto_1.1_Ls_Rest_5";
       "A0301_Fermi_P2".Sollevatori[1].DataIn.Work_Ls[1] := "A0301_CinghiaTrasporto_1.1_Ls_Work_6";
       "A0301_Fermi_P2".Sollevatori[2].DataIn.Rest_Ls[1] := "A0301_CinghiaTrasporto_2.1_Ls_Rest_5";
       "A0301_Fermi_P2".Sollevatori[2].DataIn.Work_Ls[1] := "A0301_CinghiaTrasporto_2.1_Ls_Work_6";
       "A0301_Fermi_P2".Sollevatori[3].DataIn.Rest_Ls[1] := "A0301_CinghiaTrasporto_3.1_Ls_Rest_5";
       "A0301_Fermi_P2".Sollevatori[3].DataIn.Work_Ls[1] := "A0301_CinghiaTrasporto_3.1_Ls_Work_6";
       "A0301_Fermi_P2".Sollevatori[4].DataIn.Rest_Ls[1] := "A0301_CinghiaTrasporto_4.1_Ls_Rest_5";
       "A0301_Fermi_P2".Sollevatori[4].DataIn.Work_Ls[1] := "A0301_CinghiaTrasporto_4.1_Ls_Work_6";
       "A0301_Fermi_P2".Sollevatori[5].DataIn.Rest_Ls[1] := "A0301_CinghiaTrasporto_5.1_Ls_Rest_5";
       "A0301_Fermi_P2".Sollevatori[5].DataIn.Work_Ls[1] := "A0301_CinghiaTrasporto_5.1_Ls_Work_6";
       "A0301_Fermi_P2".Sollevatori[6].DataIn.Rest_Ls[1] := "A0301_CinghiaTrasporto_6.1_Ls_Rest_5";
       "A0301_Fermi_P2".Sollevatori[6].DataIn.Work_Ls[1] := "A0301_CinghiaTrasporto_6.1_Ls_Work_6";

   END_REGION ;
END_REGION

REGION Network 3: DataIn - Fermi
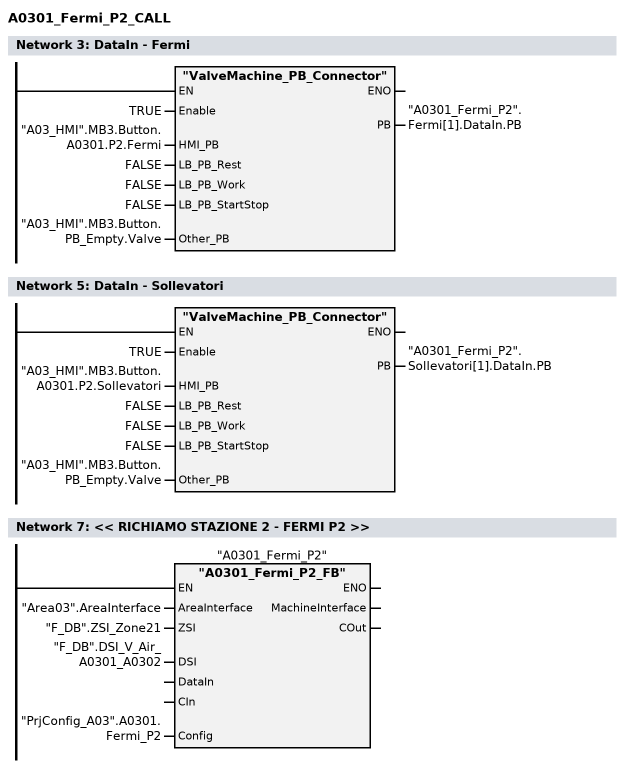
   RUNG wire#powerrail
      "ValveMachine_PB_Connector"(Enable := TRUE, HMI_PB := "A03_HMI".MB3.Button.A0301.P2.Fermi, LB_PB_Rest := FALSE, LB_PB_Work := FALSE, LB_PB_StartStop := FALSE, Other_PB := "A03_HMI".MB3.Button.PB_Empty.Valve, PB => "A0301_Fermi_P2".Fermi[1].DataIn.PB)
   END_RUNG
   // the same network as SCL:
   "ValveMachine_PB_Connector"(Enable := TRUE,
                           HMI_PB := "A03_HMI".MB3.Button.A0301.P2.Fermi,
                           LB_PB_Rest := FALSE,
                           LB_PB_Work := FALSE,
                           LB_PB_StartStop := FALSE,
                           Other_PB := "A03_HMI".MB3.Button.PB_Empty.Valve,
                           PB => "A0301_Fermi_P2".Fermi[1].DataIn.PB);
END_REGION

REGION Network 4 (SCL): DataIn - Fermi [1..6]
   // TRASFERIMENTO STATO PULSANTI - Comando manuale diretto 
   "A0301_Fermi_P2".Fermi[6].DataIn.PB := "A0301_Fermi_P2".Fermi[5].DataIn.PB := "A0301_Fermi_P2".Fermi[4].DataIn.PB :=
   "A0301_Fermi_P2".Fermi[3].DataIn.PB := "A0301_Fermi_P2".Fermi[2].DataIn.PB := "A0301_Fermi_P2".Fermi[1].DataIn.PB;
END_REGION

